C05481=1213.407,-44.587,-40.105,179.917,5.444,148.977
C05482=1213.412,-44.836,-40.092,179.914,5.443,148.977
C05483=1213.418,-45.086,-40.080,179.911,5.443,148.978
C05484=1213.422,-45.336,-40.067,179.909,5.443,148.979
C05485=1213.428,-45.586,-40.055,179.907,5.442,148.980
C05486=1213.433,-45.835,-40.043,179.904,5.442,148.980
C05487=1213.438,-46.085,-40.030,179.902,5.442,148.981
C05488=1213.443,-46.335,-40.018,179.899,5.442,148.982
C05489=1213.449,-46.584,-40.006,179.897,5.441,148.982
C05490=1213.454,-46.834,-39.994,179.894,5.442,148.983
C05491=1213.459,-47.083,-39.981,179.892,5.441,148.984
C05492=1213.464,-47.334,-39.969,179.890,5.442,148.985
C05493=1213.469,-47.583,-39.956,179.887,5.441,148.985
C05494=1213.475,-47.833,-39.944,179.885,5.440,148.986
C05495=1213.480,-48.082,-39.932,179.883,5.441,148.986
C05496=1213.485,-48.332,-39.920,179.880,5.440,148.987
C05497=1213.490,-48.602,-39.906,179.877,5.440,148.988
C05498=1213.496,-48.872,-39.894,179.874,5.440,148.989
C05499=1213.501,-49.142,-39.881,179.872,5.440,148.989
C05500=1213.507,-49.411,-39.867,179.870,5.440,148.990
C05501=1213.512,-49.662,-39.855,179.867,5.439,148.991
C05502=1213.517,-49.911,-39.843,179.865,5.439,148.992
C05503=1213.522,-50.161,-39.831,179.862,5.439,148.992
C05504=1213.527,-50.410,-39.818,179.859,5.438,148.993
C05505=1213.533,-50.660,-39.806,179.857,5.439,148.994
C05506=1213.538,-50.909,-39.794,179.855,5.438,148.994
C05507=1213.543,-51.159,-39.782,179.853,5.438,148.995
C05508=1213.548,-51.409,-39.770,179.850,5.438,148.996
C05509=1213.553,-51.658,-39.758,179.848,5.437,148.996
C05510=1213.559,-51.908,-39.746,179.846,5.438,148.997
C05511=1213.564,-52.158,-39.733,179.843,5.437,148.998
C05512=1213.568,-52.407,-39.722,179.840,5.437,148.998
C05513=1213.574,-52.657,-39.710,179.838,5.437,148.999
C05514=1213.579,-52.906,-39.698,179.836,5.437,149.000
C05515=1213.584,-53.156,-39.686,179.834,5.437,149.000
C05516=1213.590,-53.406,-39.673,179.831,5.437,149.001
C05517=1213.594,-53.655,-39.662,179.828,5.436,149.002
C05518=1213.600,-53.905,-39.650,179.827,5.436,149.002
C05519=1213.605,-54.155,-39.637,179.824,5.436,149.003
C05520=1213.610,-54.405,-39.625,179.821,5.435,149.004
C05521=1213.616,-54.654,-39.613,179.819,5.435,149.004
C05522=1213.620,-54.903,-39.601,179.817,5.435,149.005
C05523=1213.625,-55.153,-39.590,179.814,5.435,149.006
C05524=1213.631,-55.403,-39.578,179.812,5.435,149.007
C05525=1213.636,-55.653,-39.565,179.809,5.434,149.007
C05526=1213.641,-55.902,-39.554,179.807,5.435,149.008
C05527=1213.646,-56.152,-39.542,179.804,5.434,149.009
C05528=1213.651,-56.402,-39.529,179.802,5.435,149.009
C05529=1213.656,-56.651,-39.518,179.800,5.434,149.010
C05530=1213.661,-56.901,-39.506,179.797,5.433,149.011
C05531=1213.667,-57.151,-39.494,179.795,5.434,149.011
C05532=1213.672,-57.400,-39.482,179.793,5.433,149.012
C05533=1213.677,-57.650,-39.470,179.791,5.434,149.013
C05534=1213.682,-57.900,-39.459,179.788,5.433,149.013
C05535=1213.687,-58.150,-39.447,179.785,5.433,149.014
C05536=1213.692,-58.399,-39.435,179.783,5.433,149.015
C05537=1213.697,-58.649,-39.423,179.781,5.433,149.015
C05538=1213.703,-58.899,-39.411,179.778,5.433,149.016
C05539=1213.707,-59.148,-39.400,179.776,5.432,149.017
C05540=1213.713,-59.398,-39.388,179.773,5.432,149.018
C05541=1213.718,-59.648,-39.375,179.771,5.432,149.018
C05542=1213.723,-59.897,-39.364,179.769,5.432,149.019
C05543=1213.728,-60.147,-39.352,179.767,5.432,149.019
C05544=1213.734,-60.396,-39.340,179.764,5.431,149.020
C05545=1213.739,-60.646,-39.329,179.761,5.431,149.021
C05546=1213.744,-60.896,-39.317,179.759,5.431,149.022
C05547=1213.749,-61.145,-39.305,179.757,5.431,149.022
C05548=1213.754,-61.395,-39.293,179.755,5.431,149.023
C05549=1213.759,-61.645,-39.281,179.752,5.431,149.024
C05550=1213.764,-61.895,-39.270,179.749,5.430,149.024
C05551=1213.770,-62.144,-39.258,179.747,5.431,149.025
C05552=1213.775,-62.394,-39.246,179.744,5.430,149.026
C05553=1213.780,-62.644,-39.235,179.743,5.430,149.026
C05554=1213.786,-62.893,-39.224,179.740,5.430,149.027
C05555=1213.790,-63.143,-39.212,179.738,5.429,149.028
C05556=1213.796,-63.392,-39.200,179.735,5.430,149.028
C05557=1213.801,-63.642,-39.188,179.733,5.429,149.029
C05558=1213.806,-63.892,-39.176,179.731,5.429,149.030
C05559=1213.811,-64.142,-39.165,179.728,5.429,149.031
C05560=1213.816,-64.391,-39.153,179.725,5.429,149.031
C05561=1213.821,-64.641,-39.141,179.723,5.429,149.032
C05562=1213.827,-64.890,-39.131,179.721,5.428,149.033
C05563=1213.832,-65.140,-39.119,179.719,5.428,149.033
C05564=1213.837,-65.390,-39.107,179.716,5.428,149.034
C05565=1213.842,-65.640,-39.095,179.714,5.428,149.035
C05566=1213.848,-65.890,-39.084,179.712,5.428,149.035
C05567=1213.852,-66.139,-39.072,179.709,5.427,149.036
C05568=1213.858,-66.389,-39.060,179.707,5.428,149.037
C05569=1213.863,-66.638,-39.049,179.704,5.427,149.037
C05570=1213.868,-66.888,-39.038,179.702,5.428,149.038
C05571=1213.873,-67.138,-39.026,179.699,5.427,149.039
C05572=1213.878,-67.388,-39.014,179.697,5.427,149.040
C05573=1213.883,-67.637,-39.003,179.695,5.427,149.040
C05574=1213.889,-67.887,-38.991,179.692,5.426,149.041
C05575=1213.894,-68.136,-38.980,179.690,5.427,149.041
C05576=1213.899,-68.386,-38.968,179.688,5.426,149.042
C05577=1213.904,-68.636,-38.957,179.686,5.427,149.043
C05578=1213.909,-68.886,-38.945,179.683,5.426,149.044
C05579=1213.914,-69.135,-38.934,179.680,5.426,149.044
C05580=1213.920,-69.385,-38.923,179.678,5.426,149.045
C05581=1213.925,-69.635,-38.912,179.676,5.426,149.046
C05582=1213.931,-69.885,-38.900,179.673,5.426,149.046
C05583=1213.935,-70.134,-38.889,179.671,5.425,149.047
C05584=1213.941,-70.384,-38.877,179.669,5.425,149.048
C05585=1213.946,-70.633,-38.866,179.667,5.425,149.048
C05586=1213.951,-70.883,-38.855,179.664,5.425,149.049
C05587=1213.956,-71.133,-38.843,179.662,5.425,149.050
C05588=1213.961,-71.383,-38.832,179.659,5.424,149.050
C05589=1213.967,-71.632,-38.821,179.657,5.425,149.051
C05590=1213.972,-71.882,-38.809,179.654,5.424,149.052
C05591=1213.977,-72.132,-38.797,179.652,5.425,149.052
C05592=1213.982,-72.381,-38.786,179.650,5.424,149.053
C05593=1213.987,-72.630,-38.775,179.647,5.423,149.054
C05594=1213.993,-72.881,-38.764,179.645,5.424,149.054
C05595=1213.998,-73.130,-38.753,179.643,5.423,149.055
C05596=1214.003,-73.380,-38.741,179.641,5.424,149.056
C05597=1214.008,-73.629,-38.730,179.638,5.423,149.056
C05598=1214.013,-73.879,-38.719,179.636,5.424,149.057
C05599=1214.019,-74.129,-38.707,179.633,5.423,149.058
C05600=1214.024,-74.379,-38.696,179.631,5.424,149.059
C05601=1214.030,-74.649,-38.684,179.628,5.423,149.059
C05602=1214.035,-74.920,-38.671,179.626,5.423,149.060
C05603=1214.041,-75.190,-38.659,179.623,5.422,149.061
C05604=1214.046,-75.461,-38.648,179.621,5.423,149.061
C05605=1214.052,-75.711,-38.636,179.618,5.422,149.062
C05606=1214.057,-75.960,-38.626,179.616,5.422,149.063
C05607=1214.062,-76.210,-38.614,179.613,5.422,149.064
C05608=1214.067,-76.460,-38.603,179.611,5.422,149.064
C05609=1214.072,-76.709,-38.591,179.609,5.422,149.065
C05610=1214.078,-76.959,-38.581,179.607,5.421,149.065
C05611=1214.083,-77.209,-38.569,179.604,5.421,149.066
C05612=1214.088,-77.458,-38.558,179.602,5.421,149.067
C05613=1214.093,-77.708,-38.548,179.600,5.421,149.068
C05614=1214.099,-77.958,-38.536,179.597,5.421,149.068
C05615=1214.103,-78.208,-38.524,179.595,5.421,149.069
C05616=1214.109,-78.457,-38.514,179.592,5.421,149.070
C05617=1214.114,-78.707,-38.502,179.590,5.421,149.070
C05618=1214.119,-78.957,-38.491,179.588,5.420,149.071
C05619=1214.125,-79.206,-38.481,179.585,5.420,149.072
C05620=1214.129,-79.456,-38.470,179.583,5.420,149.072
C05621=1214.135,-79.706,-38.458,179.581,5.420,149.073
C05622=1214.140,-79.955,-38.447,179.579,5.420,149.074
C05623=1214.145,-80.205,-38.436,179.576,5.420,149.074
C05624=1214.150,-80.455,-38.426,179.574,5.420,149.075
C05625=1214.156,-80.704,-38.414,179.571,5.420,149.076
C05626=1214.161,-80.954,-38.403,179.569,5.420,149.076
C05627=1214.166,-81.204,-38.392,179.567,5.419,149.077
C05628=1214.171,-81.453,-38.381,179.565,5.420,149.078
C05629=1214.177,-81.704,-38.370,179.562,5.419,149.078
C05630=1214.182,-81.953,-38.359,179.559,5.419,149.079
C05631=1214.187,-82.203,-38.349,179.557,5.419,149.080
C05632=1214.192,-82.453,-38.337,179.555,5.419,149.081
C05633=1214.198,-82.702,-38.327,179.553,5.419,149.081
C05634=1214.203,-82.952,-38.315,179.550,5.418,149.082
C05635=1214.208,-83.202,-38.305,179.548,5.419,149.083
C05636=1214.213,-83.451,-38.294,179.546,5.418,149.083
C05637=1214.218,-83.701,-38.282,179.543,5.419,149.084
C05638=1214.224,-83.950,-38.272,179.541,5.418,149.085
C05639=1214.228,-84.200,-38.261,179.539,5.418,149.085
C05640=1214.234,-84.451,-38.250,179.536,5.418,149.086
C05641=1214.239,-84.699,-38.239,179.534,5.418,149.087
C05642=1214.244,-84.950,-38.228,179.532,5.418,149.087
C05643=1214.250,-85.199,-38.218,179.530,5.418,149.088
C05644=1214.255,-85.449,-38.207,179.527,5.417,149.089
C05645=1214.260,-85.699,-38.196,179.524,5.417,149.089
C05646=1214.265,-85.948,-38.185,179.522,5.417,149.090
C05647=1214.271,-86.199,-38.174,179.520,5.417,149.091
C05648=1214.276,-86.448,-38.163,179.518,5.417,149.092
C05649=1214.281,-86.698,-38.153,179.515,5.417,149.092
C05650=1214.286,-86.947,-38.142,179.513,5.417,149.093
C05651=1214.291,-87.197,-38.131,179.511,5.416,149.093
C05652=1214.296,-87.447,-38.121,179.508,5.417,149.094
C05653=1214.301,-87.696,-38.110,179.506,5.416,149.095
C05654=1214.306,-87.946,-38.099,179.504,5.417,149.096
C05655=1214.312,-88.195,-38.088,179.501,5.416,149.096
C05656=1214.317,-88.446,-38.078,179.499,5.416,149.097
C05657=1214.323,-88.695,-38.067,179.497,5.416,149.097
C05658=1214.328,-88.945,-38.055,179.495,5.416,149.098
C05659=1214.333,-89.195,-38.045,179.492,5.416,149.099
C05660=1214.338,-89.445,-38.035,179.490,5.416,149.100
C05661=1214.344,-89.694,-38.024,179.487,5.416,149.100
C05662=1214.349,-89.944,-38.013,179.485,5.416,149.101
C05663=1214.354,-90.194,-38.003,179.483,5.415,149.101
C05664=1214.359,-90.443,-37.992,179.480,5.415,149.102
C05665=1214.365,-90.693,-37.981,179.478,5.415,149.103
C05666=1214.370,-90.943,-37.971,179.476,5.415,149.104
C05667=1214.374,-91.193,-37.960,179.473,5.415,149.104
C05668=1214.380,-91.442,-37.949,179.471,5.415,149.105
C05669=1214.385,-91.692,-37.939,179.469,5.415,149.106
C05670=1214.390,-91.941,-37.928,179.466,5.414,149.106
C05671=1214.396,-92.191,-37.918,179.464,5.415,149.107
C05672=1214.401,-92.441,-37.907,179.462,5.414,149.108
C05673=1214.406,-92.691,-37.897,179.460,5.415,149.108
C05674=1214.411,-92.940,-37.886,179.457,5.414,149.109
C05675=1214.417,-93.190,-37.875,179.455,5.415,149.110
C05676=1214.422,-93.440,-37.865,179.453,5.414,149.110
C05677=1214.427,-93.690,-37.855,179.451,5.414,149.111
C05678=1214.432,-93.939,-37.843,179.448,5.414,149.112
C05679=1214.437,-94.189,-37.833,179.446,5.414,149.112
C05680=1214.442,-94.439,-37.823,179.443,5.414,149.113
C05681=1214.448,-94.689,-37.812,179.441,5.414,149.114
C05682=1214.453,-94.939,-37.802,179.439,5.413,149.114
C05683=1214.458,-95.188,-37.791,179.437,5.414,149.115
C05684=1214.463,-95.438,-37.780,179.434,5.413,149.116
C05685=1214.469,-95.687,-37.770,179.432,5.413,149.116
C05686=1214.475,-95.937,-37.760,179.429,5.413,149.117
C05687=1214.480,-96.187,-37.749,179.427,5.413,149.118
C05688=1214.485,-96.436,-37.738,179.425,5.413,149.118
C05689=1214.490,-96.686,-37.728,179.423,5.413,149.119
C05690=1214.495,-96.936,-37.718,179.420,5.413,149.120
C05691=1214.500,-97.186,-37.708,179.418,5.413,149.121
C05692=1214.505,-97.435,-37.697,179.416,5.413,149.121
C05693=1214.511,-97.685,-37.687,179.413,5.413,149.122
C05694=1214.516,-97.935,-37.677,179.411,5.412,149.122
C05695=1214.521,-98.185,-37.666,179.409,5.412,149.123
C05696=1214.526,-98.434,-37.655,179.407,5.412,149.124
C05697=1214.532,-98.684,-37.645,179.404,5.412,149.125
C05698=1214.537,-98.934,-37.635,179.402,5.412,149.125
C05699=1214.542,-99.184,-37.624,179.400,5.412,149.126
C05700=1214.547,-99.433,-37.615,179.397,5.412,149.126
C05701=1214.552,-99.683,-37.604,179.395,5.412,149.127
C05702=1214.558,-99.933,-37.594,179.393,5.411,149.128
C05703=1214.563,-100.182,-37.584,179.391,5.412,149.129
C05704=1214.568,-100.433,-37.573,179.388,5.411,149.129
C05705=1214.574,-100.704,-37.562,179.385,5.411,149.130
C05706=1214.580,-100.975,-37.551,179.383,5.411,149.131
C05707=1214.585,-101.246,-37.540,179.380,5.411,149.131
C05708=1214.591,-101.518,-37.528,179.378,5.411,149.132
C05709=1214.596,-101.767,-37.519,179.376,5.411,149.133
C05710=1214.601,-102.016,-37.508,179.374,5.411,149.134
C05711=1214.606,-102.266,-37.497,179.371,5.410,149.134
C05712=1214.612,-102.516,-37.487,179.369,5.411,149.135
C05713=1214.617,-102.766,-37.476,179.367,5.410,149.136
C05714=1214.622,-103.016,-37.468,179.365,5.411,149.136
C05715=1214.628,-103.265,-37.457,179.362,5.410,149.137
C05716=1214.633,-103.515,-37.447,179.360,5.410,149.137
C05717=1214.638,-103.765,-37.437,179.358,5.410,149.138
C05718=1214.644,-104.015,-37.426,179.356,5.410,149.139
C05719=1214.648,-104.265,-37.416,179.353,5.410,149.140
C05720=1214.654,-104.514,-37.406,179.351,5.410,149.140
C05721=1214.659,-104.764,-37.396,179.349,5.409,149.141
C05722=1214.664,-105.014,-37.385,179.347,5.410,149.141
C05723=1214.669,-105.263,-37.376,179.344,5.409,149.142
C05724=1214.675,-105.513,-37.366,179.342,5.410,149.143
C05725=1214.680,-105.763,-37.355,179.339,5.409,149.144
C05726=1214.685,-106.012,-37.345,179.337,5.409,149.144
C05727=1214.690,-106.262,-37.335,179.335,5.409,149.145
C05728=1214.696,-106.511,-37.325,179.333,5.409,149.146
C05729=1214.701,-106.762,-37.315,179.330,5.409,149.146
C05730=1214.707,-107.012,-37.305,179.328,5.409,149.147
C05731=1214.712,-107.261,-37.295,179.326,5.409,149.147
C05732=1214.717,-107.511,-37.285,179.324,5.409,149.148
C05733=1214.722,-107.761,-37.275,179.321,5.408,149.149
C05734=1214.727,-108.010,-37.265,179.319,5.409,149.150
C05735=1214.732,-108.260,-37.254,179.316,5.408,149.150
C05736=1214.738,-108.510,-37.245,179.315,5.408,149.151
C05737=1214.743,-108.759,-37.235,179.312,5.408,149.152
C05738=1214.748,-109.009,-37.225,179.310,5.408,149.152
C05739=1214.753,-109.259,-37.214,179.307,5.408,149.153
C05740=1214.759,-109.509,-37.204,179.305,5.408,149.154
C05741=1214.764,-109.758,-37.195,179.303,5.408,149.154
C05742=1214.770,-110.008,-37.185,179.301,5.408,149.155
C05743=1214.775,-110.258,-37.175,179.299,5.408,149.156
C05744=1214.780,-110.508,-37.165,179.296,5.408,149.156
C05745=1214.785,-110.757,-37.155,179.294,5.408,149.157
C05746=1214.790,-111.007,-37.146,179.292,5.407,149.157
C05747=1214.795,-111.257,-37.135,179.290,5.408,149.158
C05748=1214.801,-111.507,-37.125,179.287,5.407,149.159
C05749=1214.806,-111.756,-37.115,179.285,5.408,149.160
C05750=1214.812,-112.006,-37.106,179.283,5.407,149.160
C05751=1214.817,-112.257,-37.095,179.281,5.407,149.161
C05752=1214.822,-112.506,-37.086,179.278,5.407,149.162
C05753=1214.827,-112.755,-37.076,179.276,5.407,149.162
C05754=1214.832,-113.005,-37.067,179.273,5.407,149.163
C05755=1214.838,-113.255,-37.056,179.272,5.407,149.163
C05756=1214.843,-113.505,-37.046,179.269,5.407,149.164
C05757=1214.848,-113.755,-37.037,179.267,5.407,149.165
C05758=1214.854,-114.004,-37.027,179.264,5.407,149.166
C05759=1214.859,-114.254,-37.017,179.263,5.406,149.166
C05760=1214.864,-114.503,-37.007,179.260,5.406,149.167
C05761=1214.870,-114.754,-36.997,179.258,5.406,149.168
C05762=1214.874,-115.003,-36.987,179.255,5.406,149.168
C05763=1214.880,-115.253,-36.977,179.253,5.406,149.169
C05764=1214.885,-115.503,-36.968,179.251,5.406,149.169
C05765=1214.891,-115.752,-36.958,179.249,5.406,149.170
C05766=1214.895,-116.003,-36.949,179.247,5.406,149.171
C05767=1214.901,-116.252,-36.939,179.244,5.406,149.172
C05768=1214.907,-116.502,-36.928,179.242,5.406,149.172
C05769=1214.912,-116.752,-36.920,179.240,5.406,149.173
C05770=1214.917,-117.001,-36.909,179.238,5.406,149.173
C05771=1214.922,-117.250,-36.900,179.235,5.406,149.174
C05772=1214.927,-117.501,-36.890,179.233,5.406,149.175
C05773=1214.932,-117.750,-36.880,179.231,5.405,149.175
C05774=1214.938,-118.001,-36.871,179.229,5.406,149.176
C05775=1214.943,-118.250,-36.861,179.226,5.405,149.177
C05776=1214.949,-118.500,-36.852,179.224,5.405,149.177
C05777=1214.954,-118.749,-36.842,179.222,5.405,149.178
C05778=1214.959,-118.999,-36.832,179.219,5.405,149.179
C05779=1214.964,-119.249,-36.823,179.217,5.405,149.179
C05780=1214.970,-119.499,-36.812,179.215,5.405,149.180
C05781=1214.975,-119.749,-36.803,179.213,5.405,149.181
C05782=1214.980,-119.998,-36.793,179.210,5.405,149.181
C05783=1214.986,-120.248,-36.784,179.208,5.405,149.182
C05784=1214.990,-120.497,-36.775,179.206,5.404,149.183
C05785=1214.996,-120.748,-36.765,179.204,5.405,149.183
C05786=1215.001,-120.997,-36.755,179.201,5.404,149.184
C05787=1215.007,-121.248,-36.746,179.199,5.405,149.185
C05788=1215.011,-121.497,-36.736,179.197,5.404,149.185
C05789=1215.017,-121.747,-36.727,179.195,5.404,149.186
C05790=1215.022,-121.996,-36.717,179.192,5.404,149.187
C05791=1215.028,-122.246,-36.708,179.190,5.404,149.187
C05792=1215.033,-122.496,-36.698,179.189,5.404,149.188
C05793=1215.038,-122.746,-36.689,179.186,5.404,149.189
C05794=1215.044,-122.995,-36.679,179.184,5.404,149.189
C05795=1215.049,-123.245,-36.670,179.181,5.404,149.190
C05796=1215.054,-123.495,-36.659,179.180,5.404,149.190
C05797=1215.059,-123.745,-36.650,179.177,5.403,149.191
C05798=1215.064,-123.995,-36.642,179.175,5.404,149.192
C05799=1215.070,-124.244,-36.631,179.172,5.403,149.193
C05800=1215.075,-124.494,-36.622,179.171,5.403,149.193
C05801=1215.081,-124.744,-36.612,179.168,5.403,149.194
C05802=1215.086,-124.994,-36.603,179.166,5.403,149.195
C05803=1215.091,-125.244,-36.594,179.164,5.403,149.195
C05804=1215.096,-125.493,-36.584,179.161,5.403,149.196
C05805=1215.102,-125.743,-36.575,179.159,5.403,149.196
C05806=1215.106,-125.992,-36.566,179.157,5.403,149.197
C05807=1215.112,-126.242,-36.556,179.155,5.403,149.198
C05808=1215.118,-126.492,-36.547,179.152,5.403,149.198
C05809=1214.696,-126.503,-36.584,179.148,5.406,149.201
C05810=1214.691,-126.254,-36.593,179.151,5.406,149.200
C05811=1214.685,-126.003,-36.603,179.153,5.406,149.199
C05812=1214.680,-125.754,-36.612,179.155,5.406,149.198
C05813=1214.674,-125.504,-36.622,179.157,5.406,149.198
C05814=1214.669,-125.254,-36.631,179.160,5.407,149.197
C05815=1214.664,-125.005,-36.640,179.162,5.407,149.196
C05816=1214.658,-124.755,-36.650,179.164,5.406,149.196
C05817=1214.654,-124.504,-36.659,179.166,5.407,149.195
C05818=1214.649,-124.255,-36.669,179.168,5.407,149.195
C05819=1214.643,-124.005,-36.678,179.171,5.407,149.194
C05820=1214.638,-123.756,-36.688,179.172,5.407,149.193
C05821=1214.632,-123.506,-36.697,179.175,5.407,149.193
C05822=1214.627,-123.256,-36.706,179.177,5.407,149.192
C05823=1214.622,-123.006,-36.716,179.180,5.407,149.191
C05824=1214.616,-122.756,-36.725,179.181,5.407,149.191
C05825=1214.611,-122.507,-36.735,179.184,5.408,149.190
C05826=1214.606,-122.257,-36.745,179.186,5.407,149.189
C05827=1214.601,-122.008,-36.754,179.188,5.407,149.189
C05828=1214.596,-121.758,-36.763,179.191,5.408,149.188
C05829=1214.591,-121.508,-36.774,179.193,5.407,149.187
C05830=1214.585,-121.258,-36.783,179.195,5.408,149.187
C05831=1214.580,-121.008,-36.793,179.197,5.407,149.186
C05832=1214.575,-120.758,-36.802,179.200,5.408,149.185
C05833=1214.569,-120.509,-36.812,179.202,5.408,149.185
C05834=1214.564,-120.259,-36.821,179.204,5.408,149.184
C05835=1214.558,-120.009,-36.831,179.206,5.408,149.183
C05836=1214.553,-119.760,-36.840,179.209,5.409,149.183
C05837=1214.548,-119.509,-36.850,179.211,5.408,149.182
C05838=1214.543,-119.259,-36.859,179.213,5.409,149.181
C05839=1214.537,-119.010,-36.870,179.215,5.409,149.181
C05840=1214.532,-118.760,-36.878,179.217,5.408,149.180
C05841=1214.527,-118.511,-36.888,179.220,5.409,149.179
C05842=1214.521,-118.261,-36.898,179.222,5.408,149.179
C05843=1214.516,-118.011,-36.907,179.225,5.409,149.178
C05844=1214.511,-117.761,-36.918,179.226,5.409,149.178
C05845=1214.506,-117.511,-36.927,179.229,5.409,149.177
C05846=1214.501,-117.262,-36.937,179.231,5.409,149.176
C05847=1214.495,-117.012,-36.946,179.234,5.409,149.175
C05848=1214.490,-116.762,-36.956,179.235,5.409,149.175
C05849=1214.484,-116.513,-36.966,179.238,5.410,149.174
C05850=1214.480,-116.262,-36.975,179.240,5.409,149.173
C05851=1214.474,-116.013,-36.986,179.243,5.410,149.173
C05852=1214.469,-115.763,-36.995,179.244,5.410,149.172
C05853=1214.463,-115.513,-37.005,179.247,5.410,149.172
C05854=1214.459,-115.264,-37.014,179.249,5.410,149.171
C05855=1214.453,-115.014,-37.024,179.251,5.409,149.170
C05856=1214.448,-114.764,-37.034,179.253,5.410,149.170
C05857=1214.443,-114.514,-37.044,179.255,5.410,149.169
C05858=1214.437,-114.264,-37.053,179.258,5.410,149.168
C05859=1214.432,-114.015,-37.063,179.260,5.410,149.167
C05860=1214.426,-113.766,-37.073,179.262,5.410,149.167
C05861=1214.422,-113.515,-37.083,179.264,5.410,149.166
C05862=1214.416,-113.265,-37.093,179.267,5.410,149.166
C05863=1214.411,-113.016,-37.103,179.269,5.410,149.165
C05864=1214.406,-112.767,-37.113,179.272,5.411,149.164
C05865=1214.400,-112.516,-37.122,179.273,5.411,149.164
C05866=1214.396,-112.267,-37.132,179.276,5.411,149.163
C05867=1214.390,-112.017,-37.142,179.278,5.411,149.162
C05868=1214.384,-111.767,-37.152,179.281,5.411,149.161
C05869=1214.379,-111.518,-37.161,179.283,5.411,149.161
C05870=1214.374,-111.267,-37.172,179.285,5.411,149.160
C05871=1214.369,-111.018,-37.182,179.287,5.411,149.160
C05872=1214.364,-110.769,-37.192,179.290,5.411,149.159
C05873=1214.358,-110.518,-37.201,179.292,5.411,149.158
C05874=1214.354,-110.268,-37.211,179.294,5.412,149.158
C05875=1214.348,-110.019,-37.221,179.296,5.411,149.157
C05876=1214.342,-109.769,-37.232,179.298,5.411,149.156
C05877=1214.337,-109.520,-37.241,179.301,5.411,149.156
C05878=1214.332,-109.269,-37.251,179.303,5.412,149.155
C05879=1214.327,-109.020,-37.261,179.305,5.412,149.154
C05880=1214.322,-108.771,-37.271,179.307,5.412,149.154
C05881=1214.316,-108.521,-37.281,179.310,5.412,149.153
C05882=1214.311,-108.271,-37.292,179.312,5.412,149.152
C05883=1214.305,-108.021,-37.301,179.314,5.412,149.152
C05884=1214.301,-107.771,-37.311,179.317,5.412,149.151
C05885=1214.295,-107.522,-37.321,179.319,5.412,149.150
C05886=1214.290,-107.272,-37.332,179.321,5.412,149.150
C05887=1214.285,-107.022,-37.341,179.324,5.412,149.149
C05888=1214.279,-106.773,-37.351,179.326,5.412,149.148
C05889=1214.274,-106.523,-37.362,179.328,5.413,149.148
C05890=1214.269,-106.272,-37.372,179.330,5.413,149.147
C05891=1214.264,-106.023,-37.381,179.333,5.413,149.146
C05892=1214.259,-105.773,-37.392,179.335,5.413,149.145
C05893=1214.253,-105.523,-37.402,179.337,5.413,149.145
C05894=1214.248,-105.274,-37.412,179.339,5.413,149.144
C05895=1214.243,-105.024,-37.422,179.342,5.413,149.144
C05896=1214.238,-104.774,-37.432,179.344,5.413,149.143
C05897=1214.232,-104.525,-37.443,179.347,5.413,149.142
C05898=1214.227,-104.276,-37.452,179.348,5.413,149.142
C05899=1214.222,-104.025,-37.463,179.351,5.414,149.141
C05900=1214.217,-103.776,-37.473,179.353,5.413,149.140
C05901=1214.211,-103.526,-37.483,179.356,5.414,149.140
C05902=1214.206,-103.276,-37.494,179.358,5.414,149.139
C05903=1214.201,-103.027,-37.503,179.360,5.414,149.138
C05904=1214.196,-102.776,-37.513,179.362,5.414,149.138
C05905=1214.190,-102.526,-37.523,179.365,5.414,149.137
C05906=1214.185,-102.277,-37.534,179.367,5.414,149.136
C05907=1214.180,-102.027,-37.544,179.370,5.414,149.135
C05908=1214.175,-101.777,-37.554,179.372,5.414,149.135
C05909=1214.169,-101.528,-37.564,179.374,5.415,149.134
C05910=1214.164,-101.257,-37.576,179.376,5.414,149.134
C05911=1214.158,-100.986,-37.587,179.379,5.415,149.133
C05912=1214.152,-100.715,-37.598,179.381,5.415,149.132
C05913=1214.147,-100.443,-37.609,179.384,5.415,149.131
C05914=1214.142,-100.193,-37.620,179.386,5.415,149.131
C05915=1214.136,-99.944,-37.630,179.388,5.415,149.130
C05916=1214.130,-99.694,-37.640,179.391,5.415,149.129
C05917=1214.126,-99.444,-37.650,179.393,5.415,149.129
C05918=1214.121,-99.195,-37.660,179.396,5.415,149.128
C05919=1214.116,-98.944,-37.671,179.397,5.415,149.127
C05920=1214.110,-98.695,-37.681,179.400,5.416,149.127
C05921=1214.104,-98.445,-37.691,179.402,5.416,149.126
C05922=1214.099,-98.195,-37.702,179.405,5.416,149.125
C05923=1214.094,-97.945,-37.712,179.407,5.416,149.125
C05924=1214.089,-97.696,-37.724,179.410,5.416,149.124
C05925=1214.084,-97.447,-37.733,179.411,5.416,149.123
C05926=1214.079,-97.197,-37.743,179.414,5.416,149.123
C05927=1214.074,-96.947,-37.754,179.416,5.416,149.122
C05928=1214.068,-96.697,-37.764,179.419,5.417,149.121
C05929=1214.063,-96.447,-37.775,179.421,5.416,149.120
C05930=1214.057,-96.197,-37.785,179.423,5.417,149.120
C05931=1214.053,-95.948,-37.796,179.425,5.417,149.119
C05932=1214.047,-95.698,-37.806,179.428,5.417,149.119
C05933=1214.042,-95.449,-37.817,179.430,5.417,149.118
C05934=1214.037,-95.198,-37.827,179.432,5.417,149.117
C05935=1214.031,-94.949,-37.837,179.434,5.417,149.116
C05936=1214.026,-94.699,-37.849,179.437,5.417,149.116
C05937=1214.021,-94.450,-37.859,179.439,5.417,149.115
C05938=1214.016,-94.199,-37.870,179.441,5.418,149.115
C05939=1214.010,-93.950,-37.880,179.443,5.417,149.114
C05940=1214.005,-93.700,-37.890,179.446,5.418,149.113
C05941=1214.000,-93.451,-37.901,179.448,5.417,149.112
C05942=1213.995,-93.201,-37.912,179.451,5.418,149.112
C05943=1213.989,-92.951,-37.922,179.453,5.418,149.111
C05944=1213.984,-92.701,-37.932,179.455,5.418,149.110
C05945=1213.979,-92.452,-37.944,179.457,5.418,149.110
C05946=1213.973,-92.202,-37.954,179.460,5.418,149.109
C05947=1213.968,-91.952,-37.964,179.462,5.418,149.108
C05948=1213.963,-91.702,-37.974,179.465,5.418,149.108
C05949=1213.958,-91.453,-37.986,179.466,5.418,149.107
C05950=1213.952,-91.203,-37.996,179.469,5.419,149.106
C05951=1213.947,-90.953,-38.007,179.471,5.418,149.106
C05952=1213.942,-90.704,-38.017,179.474,5.419,149.105
C05953=1213.937,-90.454,-38.028,179.476,5.419,149.104
C05954=1213.932,-90.204,-38.038,179.479,5.419,149.104
C05955=1213.927,-89.955,-38.050,179.481,5.419,149.103
C05956=1213.921,-89.705,-38.060,179.483,5.419,149.102
C05957=1213.916,-89.455,-38.070,179.485,5.420,149.102
C05958=1213.912,-89.205,-38.082,179.488,5.419,149.101
C05959=1213.906,-88.956,-38.092,179.490,5.420,149.100
C05960=1213.901,-88.706,-38.102,179.492,5.419,149.100
C05961=1213.896,-88.457,-38.113,179.495,5.420,149.099
C05962=1213.891,-88.206,-38.124,179.497,5.420,149.098
C05963=1213.885,-87.957,-38.134,179.499,5.420,149.098
C05964=1213.880,-87.707,-38.145,179.501,5.420,149.097
C05965=1213.875,-87.458,-38.156,179.504,5.420,149.096
C05966=1213.869,-87.208,-38.168,179.506,5.420,149.096
C05967=1213.864,-86.958,-38.178,179.509,5.420,149.095
C05968=1213.859,-86.708,-38.188,179.511,5.420,149.094
C05969=1213.854,-86.458,-38.200,179.513,5.421,149.094
C05970=1213.848,-86.209,-38.210,179.515,5.420,149.093
C05971=1213.844,-85.959,-38.221,179.518,5.421,149.092
C05972=1213.838,-85.710,-38.231,179.520,5.421,149.091
C05973=1213.833,-85.460,-38.243,179.523,5.421,149.091
C05974=1213.827,-85.210,-38.253,179.525,5.421,149.090
C05975=1213.822,-84.960,-38.265,179.527,5.421,149.089
C05976=1213.817,-84.710,-38.275,179.530,5.421,149.089
C05977=1213.812,-84.461,-38.285,179.532,5.422,149.088
C05978=1213.807,-84.211,-38.297,179.534,5.422,149.087
C05979=1213.802,-83.962,-38.307,179.536,5.422,149.087
C05980=1213.797,-83.712,-38.318,179.539,5.422,149.086
C05981=1213.791,-83.461,-38.329,179.541,5.422,149.085
C05982=1213.786,-83.212,-38.340,179.544,5.422,149.085
C05983=1213.781,-82.962,-38.351,179.546,5.422,149.084
C05984=1213.776,-82.713,-38.362,179.548,5.423,149.083
C05985=1213.771,-82.464,-38.373,179.551,5.423,149.083
C05986=1213.765,-82.213,-38.384,179.553,5.423,149.082
C05987=1213.760,-81.964,-38.395,179.556,5.423,149.081
C05988=1213.755,-81.714,-38.406,179.558,5.423,149.081
C05989=1213.750,-81.464,-38.417,179.560,5.423,149.080
C05990=1213.745,-81.215,-38.427,179.562,5.423,149.079
C05991=1213.739,-80.965,-38.439,179.565,5.424,149.079
C05992=1213.734,-80.715,-38.449,179.567,5.423,149.078
C05993=1213.729,-80.466,-38.461,179.569,5.424,149.077
C05994=1213.724,-80.216,-38.472,179.571,5.423,149.077
C05995=1213.718,-79.966,-38.483,179.574,5.424,149.076
C05996=1213.713,-79.717,-38.494,179.576,5.423,149.075
C05997=1213.708,-79.466,-38.505,179.579,5.424,149.074
C05998=1213.703,-79.217,-38.516,179.581,5.424,149.074
C05999=1213.697,-78.967,-38.527,179.583,5.424,149.073
C06000=1213.692,-78.717,-38.538,179.586,5.425,149.073
C06001=1213.687,-78.468,-38.549,179.588,5.424,149.072
C06002=1213.682,-78.219,-38.560,179.591,5.425,149.071
C06003=1213.677,-77.968,-38.571,179.593,5.424,149.070
C06004=1213.671,-77.719,-38.582,179.595,5.425,149.070
C06005=1213.667,-77.470,-38.594,179.597,5.425,149.069
C06006=1213.661,-77.219,-38.605,179.600,5.425,149.068
C06007=1213.656,-76.970,-38.616,179.602,5.426,149.068
C06008=1213.651,-76.720,-38.627,179.604,5.425,149.067
C06009=1213.645,-76.470,-38.638,179.607,5.426,149.066
C06010=1213.641,-76.220,-38.649,179.609,5.426,149.066
C06011=1213.635,-75.971,-38.660,179.612,5.426,149.065
C06012=1213.630,-75.721,-38.672,179.614,5.426,149.064
C06013=1213.625,-75.471,-38.683,179.616,5.426,149.064
C06014=1213.619,-75.201,-38.695,179.619,5.426,149.063
C06015=1213.613,-74.930,-38.708,179.621,5.426,149.062
C06016=1213.608,-74.660,-38.719,179.624,5.427,149.061
C06017=1213.602,-74.390,-38.731,179.627,5.427,149.061
C06018=1213.597,-74.140,-38.743,179.629,5.427,149.060
C06019=1213.592,-73.890,-38.754,179.631,5.427,149.059
C06020=1213.586,-73.640,-38.765,179.633,5.427,149.059
C06021=1213.581,-73.391,-38.777,179.636,5.427,149.058
C06022=1213.576,-73.141,-38.788,179.638,5.427,149.057
C06023=1213.572,-72.891,-38.799,179.641,5.427,149.056
C06024=1213.566,-72.642,-38.811,179.643,5.428,149.056
C06025=1213.561,-72.392,-38.821,179.645,5.428,149.055
C06026=1213.555,-72.142,-38.833,179.648,5.428,149.055
C06027=1213.551,-71.892,-38.844,179.650,5.428,149.054
C06028=1213.545,-71.643,-38.856,179.653,5.428,149.053
C06029=1213.540,-71.393,-38.867,179.655,5.428,149.052
C06030=1213.535,-71.144,-38.878,179.657,5.428,149.052
C06031=1213.529,-70.893,-38.890,179.660,5.429,149.051
C06032=1213.524,-70.644,-38.901,179.662,5.428,149.050
C06033=1213.519,-70.394,-38.912,179.664,5.429,149.050
C06034=1213.514,-70.145,-38.924,179.666,5.429,149.049
C06035=1213.509,-69.895,-38.936,179.669,5.429,149.048
C06036=1213.503,-69.646,-38.947,179.671,5.429,149.048
C06037=1213.498,-69.396,-38.958,179.674,5.429,149.047
C06038=1213.493,-69.146,-38.970,179.676,5.430,149.046
C06039=1213.488,-68.896,-38.980,179.679,5.430,149.046
C06040=1213.483,-68.646,-38.992,179.681,5.430,149.045
C06041=1213.477,-68.397,-39.003,179.683,5.430,149.044
C06042=1213.472,-68.147,-39.015,179.686,5.430,149.043
C06043=1213.467,-67.898,-39.026,179.688,5.430,149.043
C06044=1213.462,-67.648,-39.038,179.690,5.431,149.042
C06045=1213.457,-67.398,-39.049,179.693,5.431,149.042
C06046=1213.452,-67.148,-39.061,179.695,5.431,149.041
C06047=1213.446,-66.899,-39.072,179.698,5.431,149.040
C06048=1213.441,-66.649,-39.084,179.700,5.431,149.039
C06049=1213.436,-66.400,-39.095,179.702,5.431,149.039
C06050=1213.431,-66.150,-39.107,179.705,5.432,149.038
C06051=1213.425,-65.900,-39.119,179.707,5.431,149.037
C06052=1213.421,-65.650,-39.130,179.709,5.432,149.037
C06053=1213.415,-65.401,-39.142,179.711,5.432,149.036
C06054=1213.410,-65.151,-39.153,179.714,5.432,149.035
C06055=1213.405,-64.901,-39.165,179.716,5.432,149.035
C06056=1213.400,-64.652,-39.176,179.719,5.432,149.034
C06057=1213.394,-64.402,-39.188,179.722,5.433,149.033
C06058=1213.390,-64.152,-39.200,179.724,5.432,149.033
C06059=1213.384,-63.902,-39.212,179.726,5.433,149.032
C06060=1213.378,-63.653,-39.223,179.728,5.433,149.031
C06061=1213.374,-63.403,-39.234,179.731,5.433,149.031
C06062=1213.368,-63.153,-39.246,179.733,5.434,149.030
C06063=1213.364,-62.904,-39.258,179.735,5.434,149.029
C06064=1213.358,-62.654,-39.270,179.738,5.434,149.029
C06065=1213.354,-62.405,-39.281,179.740,5.434,149.028
C06066=1213.348,-62.155,-39.293,179.743,5.434,149.027
C06067=1213.343,-61.905,-39.305,179.745,5.435,149.027
C06068=1213.338,-61.655,-39.316,179.747,5.434,149.026
C06069=1213.332,-61.406,-39.328,179.750,5.435,149.025
C06070=1213.327,-61.156,-39.340,179.752,5.434,149.024
C06071=1213.322,-60.907,-39.351,179.755,5.435,149.024
C06072=1213.317,-60.657,-39.364,179.758,5.435,149.023
C06073=1213.312,-60.408,-39.375,179.759,5.435,149.023
C06074=1213.307,-60.158,-39.387,179.762,5.436,149.022
C06075=1213.301,-59.908,-39.399,179.764,5.435,149.021
C06076=1213.297,-59.658,-39.410,179.767,5.436,149.020
C06077=1213.291,-59.408,-39.422,179.769,5.436,149.020
C06078=1213.286,-59.159,-39.435,179.771,5.436,149.019
C06079=1213.281,-58.909,-39.446,179.774,5.436,149.018
C06080=1213.276,-58.659,-39.458,179.776,5.436,149.018
C06081=1213.271,-58.409,-39.470,179.779,5.436,149.017
C06082=1213.265,-58.160,-39.481,179.781,5.437,149.016
C06083=1213.260,-57.911,-39.493,179.783,5.437,149.015
C06084=1213.255,-57.661,-39.505,179.786,5.437,149.015
C06085=1213.250,-57.412,-39.516,179.788,5.437,149.014
C06086=1213.245,-57.162,-39.528,179.790,5.438,149.014
C06087=1213.239,-56.912,-39.541,179.793,5.438,149.013
C06088=1213.234,-56.662,-39.553,179.795,5.438,149.012
C06089=1213.229,-56.413,-39.564,179.798,5.438,149.011
C06090=1213.224,-56.163,-39.577,179.800,5.438,149.011
C06091=1213.219,-55.913,-39.589,179.803,5.438,149.010
C06092=1213.213,-55.664,-39.600,179.805,5.439,149.009
C06093=1213.209,-55.414,-39.612,179.807,5.438,149.009
C06094=1213.204,-55.165,-39.624,179.810,5.439,149.008
C06095=1213.198,-54.915,-39.636,179.812,5.439,149.007
C06096=1213.193,-54.665,-39.647,179.814,5.439,149.007
C06097=1213.188,-54.416,-39.660,179.817,5.440,149.006
C06098=1213.183,-54.166,-39.672,179.819,5.439,149.005
C06099=1213.177,-53.916,-39.684,179.822,5.440,149.005
C06100=1213.172,-53.667,-39.696,179.824,5.440,149.004
C06101=1213.168,-53.417,-39.708,179.826,5.440,149.003
C06102=1213.162,-53.167,-39.720,179.829,5.440,149.003
C06103=1213.157,-52.918,-39.732,179.831,5.440,149.002
C06104=1213.152,-52.668,-39.744,179.834,5.441,149.001
C06105=1213.147,-52.419,-39.756,179.837,5.441,149.000
C06106=1213.142,-52.169,-39.768,179.839,5.441,149.000
C06107=1213.136,-51.919,-39.780,179.841,5.442,148.999
C06108=1213.131,-51.669,-39.792,179.843,5.442,148.999
C06109=1213.126,-51.420,-39.804,179.846,5.442,148.998
C06110=1213.121,-51.170,-39.817,179.848,5.442,148.997
C06111=1213.117,-50.920,-39.829,179.850,5.442,148.996
C06112=1213.111,-50.670,-39.841,179.853,5.442,148.996
C06113=1213.106,-50.421,-39.853,179.856,5.443,148.995
C06114=1213.101,-50.171,-39.865,179.858,5.442,148.994
C06115=1213.096,-49.921,-39.878,179.860,5.443,148.994
C06116=1213.090,-49.671,-39.889,179.863,5.443,148.993
C06117=1213.085,-49.422,-39.902,179.865,5.443,148.992
C06118=1213.080,-49.152,-39.915,179.868,5.443,148.992
C06119=1213.074,-48.882,-39.928,179.870,5.444,148.991
C06120=1213.069,-48.612,-39.941,179.873,5.444,148.990
C06121=1213.063,-48.343,-39.954,179.875,5.444,148.989
C06122=1213.058,-48.093,-39.967,179.878,5.444,148.989
C06123=1213.053,-47.843,-39.979,179.881,5.445,148.988
C06124=1213.048,-47.593,-39.991,179.883,5.445,148.987
C06125=1213.042,-47.344,-40.003,179.885,5.445,148.987
C06126=1213.037,-47.094,-40.016,179.887,5.445,148.986
C06127=1213.032,-46.844,-40.028,179.890,5.445,148.985
C06128=1213.027,-46.595,-40.040,179.893,5.446,148.984
C06129=1213.021,-46.345,-40.052,179.895,5.445,148.984
C06130=1213.016,-46.096,-40.065,179.897,5.446,148.983
C06131=1213.011,-45.846,-40.077,179.900,5.447,148.983
C06132=1213.006,-45.596,-40.090,179.902,5.446,148.982
C06133=1213.001,-45.346,-40.102,179.904,5.447,148.981
C06134=1212.996,-45.097,-40.114,179.907,5.447,148.981
C06135=1212.991,-44.848,-40.126,179.909,5.447,148.980
C06136=1212.986,-44.598,-40.139,179.912,5.447,148.979
C06137=1212.981,-44.348,-40.151,179.914,5.448,148.978
C06138=1212.976,-44.099,-40.163,179.917,5.447,148.978
C06139=1212.971,-43.848,-40.176,179.919,5.448,148.977
C06140=1212.966,-43.599,-40.188,179.921,5.448,148.976
C06141=1212.960,-43.350,-40.201,179.924,5.448,148.976
C06142=1212.955,-43.100,-40.213,179.927,5.449,148.975
C06143=1212.950,-42.850,-40.225,179.928,5.449,148.974
C06144=1212.945,-42.601,-40.238,179.931,5.449,148.974
C06145=1212.939,-42.351,-40.250,179.934,5.450,148.973
C06146=1212.935,-42.101,-40.263,179.936,5.449,148.972
C06147=1212.930,-41.852,-40.275,179.938,5.450,148.972
C06148=1212.924,-41.602,-40.287,179.941,5.450,148.971
C06149=1212.919,-41.353,-40.300,179.943,5.450,148.970
C06150=1212.913,-41.103,-40.313,179.946,5.450,148.970
C06151=1212.909,-40.853,-40.326,179.948,5.451,148.969
C06152=1212.903,-40.603,-40.338,179.950,5.450,148.968
C06153=1212.898,-40.354,-40.350,179.953,5.451,148.967
C06154=1212.893,-40.104,-40.363,179.956,5.451,148.967
C06155=1212.888,-39.855,-40.376,179.958,5.451,148.966
C06156=1212.883,-39.604,-40.388,179.960,5.452,148.966
C06157=1212.878,-39.355,-40.400,179.963,5.452,148.965
C06158=1212.873,-39.106,-40.413,179.965,5.452,148.964
C06159=1212.868,-38.856,-40.426,179.967,5.452,148.963
C06160=1212.862,-38.607,-40.438,179.970,5.453,148.963
C06161=1212.858,-38.356,-40.450,179.972,5.453,148.962
C06162=1212.852,-38.107,-40.464,179.975,5.453,148.961
C06163=1212.847,-37.858,-40.476,179.977,5.454,148.961
C06164=1212.842,-37.608,-40.489,179.980,5.453,148.960
C06165=1212.837,-37.359,-40.501,179.982,5.454,148.959
C06166=1212.832,-37.108,-40.514,179.985,5.454,148.959
C06167=1212.827,-36.859,-40.526,179.987,5.454,148.958
C06168=1212.821,-36.610,-40.539,179.990,5.454,148.957
C06169=1212.816,-36.360,-40.552,179.992,5.455,148.956
C06170=1212.811,-36.110,-40.565,179.994,5.455,148.956
C06171=1212.806,-35.861,-40.578,179.997,5.455,148.955
C06172=1212.801,-35.611,-40.590,179.999,5.456,148.955
C06173=1212.795,-35.361,-40.602,-179.999,5.455,148.954
C06174=1212.791,-35.111,-40.615,-179.996,5.456,148.953
C06175=1212.786,-34.862,-40.628,-179.993,5.456,148.952
C06176=1212.780,-34.612,-40.641,-179.991,5.456,148.952
C06177=1212.775,-34.362,-40.654,-179.989,5.457,148.951
C06178=1212.770,-34.113,-40.667,-179.986,5.457,148.950
C06179=1212.765,-33.864,-40.679,-179.983,5.458,148.950
C06180=1212.760,-33.614,-40.692,-179.981,5.457,148.949
C06181=1212.755,-33.364,-40.705,-179.979,5.458,148.948
C06182=1212.750,-33.115,-40.718,-179.976,5.458,148.948
C06183=1212.745,-32.866,-40.730,-179.974,5.458,148.947
C06184=1212.740,-32.615,-40.743,-179.972,5.459,148.946
C06185=1212.734,-32.366,-40.757,-179.969,5.459,148.946
C06186=1212.729,-32.117,-40.769,-179.967,5.459,148.945
C06187=1212.724,-31.867,-40.782,-179.964,5.459,148.944
C06188=1212.719,-31.617,-40.795,-179.962,5.460,148.944
C06189=1212.714,-31.368,-40.808,-179.960,5.459,148.943
C06190=1212.708,-31.118,-40.821,-179.957,5.460,148.942
C06191=1212.704,-30.868,-40.834,-179.954,5.460,148.942
C06192=1212.699,-30.619,-40.846,-179.952,5.460,148.941
C06193=1212.693,-30.369,-40.859,-179.949,5.461,148.940
C06194=1212.688,-30.119,-40.872,-179.947,5.461,148.939
C06195=1212.683,-29.870,-40.885,-179.944,5.462,148.939
C06196=1212.678,-29.621,-40.898,-179.943,5.462,148.938
C06197=1212.673,-29.370,-40.911,-179.940,5.462,148.938
C06198=1212.668,-29.121,-40.924,-179.937,5.463,148.937
C06199=1212.663,-28.871,-40.937,-179.935,5.462,148.936
C06200=1212.657,-28.621,-40.950,-179.932,5.463,148.935
C06201=1212.652,-28.372,-40.962,-179.930,5.463,148.935
C06202=1212.648,-28.122,-40.975,-179.928,5.463,148.934
C06203=1212.642,-27.873,-40.989,-179.925,5.463,148.933
C06204=1212.637,-27.624,-41.002,-179.922,5.464,148.933
C06205=1212.632,-27.374,-41.015,-179.920,5.464,148.932
C06206=1212.627,-27.124,-41.028,-179.918,5.464,148.931
C06207=1212.622,-26.874,-41.041,-179.915,5.464,148.931
C06208=1212.617,-26.625,-41.054,-179.912,5.465,148.930
C06209=1212.611,-26.375,-41.067,-179.911,5.465,148.929
C06210=1212.607,-26.126,-41.081,-179.908,5.465,148.929
C06211=1212.602,-25.876,-41.093,-179.905,5.466,148.928
C06212=1212.597,-25.626,-41.107,-179.903,5.466,148.927
C06213=1212.591,-25.377,-41.119,-179.901,5.466,148.927
C06214=1212.586,-25.127,-41.133,-179.898,5.467,148.926
C06215=1212.581,-24.877,-41.145,-179.895,5.467,148.925
C06216=1212.576,-24.628,-41.159,-179.893,5.467,148.925
C06217=1212.571,-24.378,-41.172,-179.891,5.467,148.924
C06218=1212.566,-24.129,-41.185,-179.888,5.468,148.923
C06219=1212.561,-23.879,-41.198,-179.885,5.468,148.922
C06220=1212.556,-23.630,-41.212,-179.883,5.468,148.922
C06221=1212.551,-23.380,-41.224,-179.881,5.468,148.921
C06222=1212.545,-23.110,-41.239,-179.878,5.469,148.920
C06223=1212.539,-22.841,-41.254,-179.875,5.469,148.920
C06224=1212.534,-22.572,-41.267,-179.873,5.470,148.919
C06225=1212.528,-22.302,-41.282,-179.871,5.470,148.918
C06226=1212.524,-22.052,-41.295,-179.868,5.470,148.918
C06227=1212.518,-21.803,-41.308,-179.865,5.471,148.917
C06228=1212.514,-21.553,-41.322,-179.863,5.471,148.916
C06229=1212.508,-21.304,-41.335,-179.860,5.471,148.916
C06230=1212.503,-21.054,-41.348,-179.858,5.471,148.915
C06231=1212.498,-20.804,-41.361,-179.855,5.472,148.914
C06232=1212.493,-20.555,-41.375,-179.852,5.472,148.913
C06233=1212.487,-20.305,-41.388,-179.850,5.472,148.913
C06234=1212.483,-20.056,-41.401,-179.848,5.473,148.912
C06235=1212.477,-19.806,-41.415,-179.846,5.473,148.912
C06236=1212.472,-19.557,-41.428,-179.843,5.474,148.911
C06237=1212.467,-19.307,-41.442,-179.841,5.473,148.910
C06238=1212.462,-19.058,-41.454,-179.838,5.474,148.909
C06239=1212.457,-18.807,-41.468,-179.836,5.474,148.909
C06240=1212.452,-18.559,-41.481,-179.833,5.474,148.908
C06241=1212.447,-18.308,-41.495,-179.831,5.474,148.907
C06242=1212.442,-18.060,-41.508,-179.828,5.475,148.907
C06243=1212.437,-17.809,-41.522,-179.825,5.475,148.906
C06244=1212.432,-17.560,-41.534,-179.823,5.475,148.905
C06245=1212.427,-17.310,-41.549,-179.821,5.476,148.905
C06246=1212.421,-17.061,-41.562,-179.818,5.476,148.904
C06247=1212.417,-16.811,-41.576,-179.816,5.477,148.903
C06248=1212.411,-16.562,-41.589,-179.814,5.477,148.903
C06249=1212.407,-16.312,-41.602,-179.811,5.477,148.902
C06250=1212.401,-16.062,-41.616,-179.809,5.478,148.901
C06251=1212.396,-15.813,-41.629,-179.806,5.478,148.901
C06252=1212.391,-15.563,-41.643,-179.804,5.478,148.900
C06253=1212.386,-15.314,-41.657,-179.801,5.478,148.899
C06254=1212.381,-15.064,-41.670,-179.798,5.479,148.899
C06255=1212.376,-14.815,-41.684,-179.796,5.479,148.898
C06256=1212.371,-14.565,-41.697,-179.794,5.479,148.897
C06257=1212.365,-14.316,-41.711,-179.791,5.480,148.897
C06258=1212.360,-14.066,-41.724,-179.788,5.480,148.896
C06259=1212.356,-13.816,-41.738,-179.786,5.481,148.895
C06260=1212.350,-13.567,-41.751,-179.784,5.481,148.895
C06261=1212.345,-13.317,-41.765,-179.782,5.481,148.894
C06262=1212.340,-13.067,-41.778,-179.779,5.482,148.893
C06263=1212.335,-12.818,-41.792,-179.776,5.482,148.893
C06264=1212.330,-12.569,-41.806,-179.774,5.482,148.892
C06265=1212.325,-12.319,-41.819,-179.771,5.482,148.891
C06266=1212.320,-12.069,-41.833,-179.769,5.483,148.891
C06267=1212.314,-11.819,-41.846,-179.766,5.483,148.890
C06268=1212.310,-11.570,-41.860,-179.764,5.484,148.889
C06269=1212.304,-11.321,-41.874,-179.761,5.483,148.888
C06270=1212.299,-11.071,-41.888,-179.759,5.484,148.888
C06271=1212.295,-10.821,-41.901,-179.757,5.485,148.887
C06272=1212.289,-10.572,-41.915,-179.754,5.485,148.887
C06273=1212.284,-10.322,-41.929,-179.752,5.485,148.886
C06274=1212.280,-10.073,-41.942,-179.749,5.485,148.885
C06275=1212.274,-9.823,-41.956,-179.747,5.486,148.885
C06276=1212.269,-9.573,-41.970,-179.744,5.486,148.884
C06277=1212.264,-9.324,-41.984,-179.742,5.486,148.883
C06278=1212.259,-9.075,-41.998,-179.739,5.487,148.882
C06279=1212.254,-8.824,-42.011,-179.737,5.487,148.882
C06280=1212.249,-8.575,-42.025,-179.734,5.488,148.881
C06281=1212.244,-8.326,-42.039,-179.731,5.488,148.880
C06282=1212.239,-8.076,-42.052,-179.729,5.488,148.880
C06283=1212.233,-7.827,-42.066,-179.727,5.489,148.879
C06284=1212.229,-7.577,-42.080,-179.724,5.489,148.879
C06285=1212.224,-7.327,-42.095,-179.722,5.490,148.878
C06286=1212.218,-7.078,-42.107,-179.720,5.489,148.877
C06287=1212.214,-6.828,-42.122,-179.717,5.490,148.876
C06288=1212.209,-6.579,-42.136,-179.714,5.490,148.876
C06289=1212.203,-6.330,-42.150,-179.712,5.491,148.875
C06290=1212.198,-6.079,-42.163,-179.709,5.491,148.874
C06291=1212.194,-5.830,-42.177,-179.707,5.491,148.874
C06292=1212.188,-5.581,-42.191,-179.704,5.492,148.873
C06293=1212.183,-5.331,-42.205,-179.702,5.492,148.872
C06294=1212.178,-5.081,-42.219,-179.699,5.493,148.872
C06295=1212.173,-4.831,-42.233,-179.697,5.493,148.871
C06296=1212.167,-4.582,-42.247,-179.695,5.493,148.870
C06297=1212.163,-4.333,-42.261,-179.692,5.494,148.870
C06298=1212.158,-4.083,-42.275,-179.689,5.494,148.869
C06299=1212.153,-3.834,-42.289,-179.687,5.495,148.868
C06300=1212.148,-3.584,-42.303,-179.684,5.495,148.868
C06301=1212.143,-3.334,-42.317,-179.682,5.495,148.867
C06302=1212.137,-3.084,-42.331,-179.679,5.495,148.866
C06303=1212.132,-2.835,-42.345,-179.677,5.496,148.866
C06304=1212.128,-2.586,-42.359,-179.674,5.496,148.865
C06305=1212.123,-2.336,-42.373,-179.672,5.497,148.865
C06306=1212.118,-2.086,-42.387,-179.670,5.497,148.864
C06307=1212.112,-1.837,-42.401,-179.667,5.497,148.863
C06308=1212.107,-1.588,-42.415,-179.664,5.498,148.862
C06309=1212.102,-1.338,-42.430,-179.662,5.498,148.862
C06310=1212.097,-1.088,-42.444,-179.659,5.499,148.861
C06311=1212.092,-0.839,-42.458,-179.657,5.499,148.860
C06312=1212.087,-0.589,-42.472,-179.654,5.499,148.860
C06313=1212.082,-0.340,-42.486,-179.652,5.500,148.859
C06314=1212.077,-0.090,-42.501,-179.649,5.500,148.858
C06315=1212.072,0.159,-42.514,-179.647,5.501,148.858
C06316=1212.067,0.408,-42.528,-179.645,5.501,148.857
C06317=1212.062,0.658,-42.542,-179.642,5.501,148.856
C06318=1212.057,0.908,-42.557,-179.640,5.502,148.856
C06319=1212.052,1.157,-42.571,-179.637,5.502,148.855
C06320=1212.047,1.406,-42.585,-179.634,5.503,148.854
C06321=1212.042,1.656,-42.599,-179.632,5.503,148.854
C06322=1212.037,1.906,-42.613,-179.630,5.503,148.853
C06323=1212.032,2.156,-42.628,-179.627,5.503,148.852
C06324=1212.027,2.405,-42.642,-179.624,5.504,148.852
C06325=1212.021,2.654,-42.656,-179.622,5.505,148.851
C06326=1212.016,2.924,-42.671,-179.619,5.505,148.850
C06327=1212.011,3.193,-42.687,-179.616,5.505,148.850
C06328=1212.005,3.462,-42.702,-179.614,5.506,148.849
C06329=1211.999,3.731,-42.718,-179.611,5.506,148.848
C06330=1211.994,3.981,-42.732,-179.609,5.506,148.848
C06331=1211.989,4.230,-42.746,-179.606,5.507,148.847
C06332=1211.984,4.480,-42.760,-179.604,5.507,148.846
C06333=1211.979,4.729,-42.775,-179.601,5.508,148.845
C06334=1211.974,4.979,-42.789,-179.599,5.509,148.845
C06335=1211.969,5.228,-42.804,-179.596,5.509,148.844
C06336=1211.964,5.478,-42.818,-179.594,5.509,148.844
C06337=1211.959,5.727,-42.832,-179.591,5.509,148.843
C06338=1211.954,5.976,-42.846,-179.589,5.510,148.842
C06339=1211.949,6.226,-42.861,-179.586,5.510,148.842
C06340=1211.944,6.476,-42.875,-179.583,5.511,148.841
C06341=1211.939,6.725,-42.890,-179.581,5.511,148.840
C06342=1211.934,6.975,-42.904,-179.578,5.512,148.840
C06343=1211.929,7.225,-42.919,-179.577,5.512,148.839
C06344=1211.924,7.474,-42.933,-179.574,5.512,148.838
C06345=1211.919,7.724,-42.948,-179.571,5.513,148.838
C06346=1211.914,7.973,-42.962,-179.569,5.513,148.837
C06347=1211.909,8.222,-42.977,-179.566,5.514,148.836
C06348=1211.904,8.472,-42.991,-179.563,5.515,148.836
C06349=1211.899,8.722,-43.005,-179.561,5.514,148.835
C06350=1211.894,8.971,-43.020,-179.559,5.515,148.834
C06351=1211.888,9.221,-43.035,-179.556,5.515,148.834
C06352=1211.883,9.470,-43.049,-179.554,5.516,148.833
C06353=1211.878,9.720,-43.064,-179.551,5.517,148.832
C06354=1211.874,9.969,-43.079,-179.548,5.517,148.832
C06355=1211.869,10.219,-43.093,-179.546,5.518,148.831
C06356=1211.864,10.469,-43.107,-179.544,5.517,148.830
C06357=1211.858,10.717,-43.122,-179.541,5.518,148.830
C06358=1211.853,10.967,-43.137,-179.538,5.518,148.829
C06359=1211.848,11.217,-43.151,-179.536,5.519,148.828
C06360=1211.843,11.466,-43.166,-179.533,5.519,148.828
C06361=1211.838,11.716,-43.180,-179.531,5.520,148.827
C06362=1211.833,11.966,-43.195,-179.528,5.521,148.826
C06363=1211.828,12.215,-43.210,-179.526,5.521,148.826
C06364=1211.823,12.464,-43.224,-179.524,5.521,148.825
C06365=1211.818,12.714,-43.239,-179.521,5.522,148.824
C06366=1211.813,12.963,-43.254,-179.518,5.522,148.824
C06367=1211.808,13.213,-43.268,-179.516,5.523,148.823
C06368=1211.803,13.462,-43.283,-179.513,5.523,148.822
C06369=1211.798,13.712,-43.298,-179.510,5.524,148.822
C06370=1211.794,13.961,-43.313,-179.508,5.525,148.821
C06371=1211.788,14.211,-43.328,-179.506,5.524,148.821
C06372=1211.783,14.461,-43.342,-179.504,5.525,148.820
C06373=1211.778,14.710,-43.357,-179.501,5.525,148.819
C06374=1211.773,14.960,-43.371,-179.498,5.526,148.818
C06375=1211.768,15.209,-43.387,-179.496,5.526,148.818
C06376=1211.763,15.459,-43.401,-179.493,5.527,148.817
C06377=1211.758,15.708,-43.416,-179.490,5.527,148.816
C06378=1211.753,15.958,-43.431,-179.488,5.528,148.816
C06379=1211.748,16.207,-43.446,-179.486,5.528,148.815
C06380=1211.743,16.457,-43.460,-179.483,5.528,148.815
C06381=1211.738,16.706,-43.476,-179.481,5.529,148.814
C06382=1211.733,16.956,-43.490,-179.478,5.529,148.813
C06383=1211.728,17.205,-43.505,-179.475,5.530,148.813
C06384=1211.722,17.455,-43.520,-179.473,5.531,148.812
C06385=1211.718,17.704,-43.535,-179.470,5.531,148.811
C06386=1211.713,17.954,-43.549,-179.468,5.532,148.811
C06387=1211.707,18.203,-43.565,-179.466,5.532,148.810
C06388=1211.702,18.453,-43.579,-179.463,5.532,148.809
C06389=1211.698,18.702,-43.594,-179.461,5.533,148.809
C06390=1211.692,18.951,-43.610,-179.458,5.533,148.808
C06391=1211.687,19.201,-43.624,-179.455,5.534,148.807
C06392=1211.683,19.450,-43.639,-179.453,5.534,148.807
C06393=1211.678,19.701,-43.654,-179.451,5.535,148.806
C06394=1211.673,19.950,-43.669,-179.448,5.536,148.806
C06395=1211.668,20.199,-43.685,-179.445,5.536,148.805
C06396=1211.663,20.449,-43.699,-179.443,5.537,148.804
C06397=1211.658,20.698,-43.714,-179.441,5.536,148.803
C06398=1211.653,20.948,-43.729,-179.438,5.537,148.803
C06399=1211.648,21.197,-43.744,-179.435,5.537,148.802
C06400=1211.642,21.447,-43.759,-179.433,5.538,148.801
C06401=1211.638,21.696,-43.774,-179.430,5.539,148.801
C06402=1211.633,21.945,-43.789,-179.428,5.539,148.800
C06403=1211.627,22.195,-43.804,-179.425,5.540,148.800
C06404=1211.623,22.445,-43.820,-179.422,5.540,148.799
C06405=1211.618,22.695,-43.834,-179.420,5.541,148.798
C06406=1211.613,22.944,-43.849,-179.417,5.541,148.798
C06407=1211.607,23.193,-43.865,-179.415,5.542,148.797
C06408=1211.603,23.442,-43.880,-179.413,5.542,148.796
C06409=1211.597,23.692,-43.895,-179.410,5.543,148.796
C06410=1211.592,23.941,-43.910,-179.408,5.543,148.795
C06411=1211.587,24.191,-43.925,-179.405,5.544,148.794
C06412=1211.583,24.441,-43.941,-179.402,5.544,148.794
C06413=1211.577,24.691,-43.956,-179.400,5.545,148.793
C06414=1211.573,24.940,-43.971,-179.397,5.545,148.792
C06415=1211.567,25.189,-43.986,-179.395,5.546,148.792
C06416=1211.563,25.438,-44.001,-179.392,5.547,148.791
C06417=1211.557,25.688,-44.016,-179.390,5.547,148.791
C06418=1211.552,25.937,-44.031,-179.387,5.548,148.790
C06419=1211.548,26.187,-44.047,-179.384,5.548,148.789
C06420=1211.543,26.437,-44.062,-179.382,5.548,148.789
C06421=1211.538,26.686,-44.078,-179.380,5.548,148.788
C06422=1211.533,26.935,-44.093,-179.377,5.549,148.787
C06423=1211.527,27.185,-44.108,-179.375,5.550,148.787
C06424=1211.522,27.434,-44.123,-179.372,5.550,148.786
C06425=1211.518,27.684,-44.138,-179.370,5.551,148.785
C06426=1211.512,27.934,-44.154,-179.367,5.552,148.785
C06427=1211.508,28.183,-44.169,-179.364,5.552,148.784
C06428=1211.502,28.432,-44.185,-179.362,5.553,148.784
C06429=1211.498,28.681,-44.200,-179.359,5.553,148.783
C06430=1211.492,28.951,-44.216,-179.357,5.554,148.782
C06431=1211.487,29.219,-44.233,-179.354,5.555,148.782
C06432=1211.482,29.488,-44.250,-179.352,5.555,148.781
C06433=1211.476,29.757,-44.266,-179.348,5.555,148.780
C06434=1211.471,30.006,-44.282,-179.346,5.556,148.779
C06435=1211.466,30.255,-44.297,-179.344,5.557,148.779
C06436=1211.461,30.505,-44.312,-179.341,5.557,148.778
C06437=1211.456,30.755,-44.328,-179.338,5.558,148.777
C06438=1211.451,31.004,-44.343,-179.336,5.558,148.777
C06439=1211.446,31.253,-44.359,-179.333,5.559,148.776
C06440=1211.441,31.503,-44.374,-179.331,5.560,148.776
C06441=1211.436,31.752,-44.390,-179.328,5.560,148.775
C06442=1211.431,32.002,-44.405,-179.326,5.561,148.774
C06443=1211.426,32.251,-44.421,-179.323,5.561,148.774
C06444=1211.421,32.500,-44.436,-179.320,5.562,148.773
C06445=1211.416,32.750,-44.452,-179.318,5.562,148.772
C06446=1211.411,33.000,-44.467,-179.315,5.563,148.772
C06447=1211.406,33.249,-44.482,-179.313,5.564,148.771
C06448=1211.401,33.499,-44.498,-179.310,5.564,148.770
C06449=1211.396,33.748,-44.514,-179.308,5.564,148.770
C06450=1211.391,33.998,-44.529,-179.306,5.565,148.769
C06451=1211.386,34.247,-44.545,-179.303,5.565,148.768
C06452=1211.382,34.496,-44.561,-179.301,5.566,148.768
C06453=1211.376,34.746,-44.577,-179.298,5.567,148.767
C06454=1211.372,34.995,-44.592,-179.295,5.567,148.767
C06455=1211.367,35.245,-44.608,-179.293,5.568,148.766
C06456=1211.361,35.494,-44.623,-179.290,5.568,148.765
C06457=1211.356,35.744,-44.639,-179.287,5.569,148.765
C06458=1211.352,35.994,-44.654,-179.285,5.570,148.764
C06459=1211.347,36.243,-44.670,-179.283,5.570,148.763
C06460=1211.341,36.492,-44.686,-179.280,5.571,148.763
C06461=1211.336,36.741,-44.702,-179.277,5.571,148.762
C06462=1211.331,36.991,-44.718,-179.275,5.572,148.761
C06463=1211.327,37.240,-44.733,-179.272,5.572,148.761
C06464=1211.321,37.490,-44.748,-179.270,5.573,148.760
C06465=1211.317,37.739,-44.765,-179.267,5.574,148.760
C06466=1211.311,37.989,-44.781,-179.265,5.574,148.759
C06467=1211.306,38.238,-44.796,-179.262,5.575,148.758
C06468=1211.302,38.488,-44.811,-179.259,5.575,148.758
C06469=1211.297,38.737,-44.827,-179.257,5.576,148.757
C06470=1211.292,38.987,-44.844,-179.255,5.577,148.757
C06471=1211.287,39.236,-44.859,-179.252,5.577,148.756
C06472=1211.281,39.486,-44.875,-179.249,5.578,148.755
C06473=1211.276,39.736,-44.891,-179.247,5.578,148.755
C06474=1211.272,39.984,-44.907,-179.244,5.579,148.754
C06475=1211.267,40.234,-44.922,-179.242,5.580,148.753
C06476=1211.262,40.484,-44.938,-179.239,5.580,148.753
C06477=1211.257,40.732,-44.954,-179.237,5.581,148.752
C06478=1211.252,40.983,-44.970,-179.234,5.581,148.751
C06479=1211.247,41.232,-44.986,-179.231,5.582,148.751
C06480=1211.242,41.481,-45.002,-179.229,5.583,148.750
C06481=1211.237,41.731,-45.018,-179.227,5.583,148.750
C06482=1211.231,41.980,-45.034,-179.224,5.584,148.749
C06483=1211.227,42.230,-45.050,-179.221,5.584,148.748
C06484=1211.222,42.479,-45.065,-179.219,5.585,148.748
C06485=1211.217,42.728,-45.081,-179.216,5.586,148.747
C06486=1211.212,42.978,-45.098,-179.214,5.586,148.746
C06487=1211.207,43.227,-45.113,-179.211,5.587,148.746
C06488=1211.203,43.477,-45.130,-179.209,5.588,148.745
C06489=1211.197,43.726,-45.146,-179.206,5.588,148.744
C06490=1211.192,43.976,-45.162,-179.204,5.589,148.744
C06491=1211.187,44.225,-45.178,-179.201,5.590,148.743
C06492=1211.182,44.474,-45.193,-179.199,5.590,148.743
C06493=1211.177,44.724,-45.210,-179.196,5.591,148.742
C06494=1211.172,44.973,-45.226,-179.193,5.591,148.741
C06495=1211.168,45.223,-45.242,-179.191,5.592,148.741
C06496=1211.162,45.472,-45.258,-179.188,5.593,148.740
C06497=1211.157,45.722,-45.274,-179.186,5.593,148.740
C06498=1211.152,45.971,-45.290,-179.183,5.594,148.739
C06499=1211.148,46.221,-45.306,-179.181,5.594,148.738
C06500=1211.143,46.470,-45.322,-179.178,5.595,148.738
C06501=1211.138,46.720,-45.338,-179.176,5.596,148.737
C06502=1211.133,46.969,-45.355,-179.173,5.596,148.736
C06503=1211.128,47.219,-45.371,-179.170,5.597,148.736
C06504=1211.123,47.468,-45.387,-179.168,5.597,148.735
C06505=1211.118,47.717,-45.404,-179.166,5.598,148.735
C06506=1211.113,47.966,-45.419,-179.163,5.599,148.734
C06507=1211.108,48.216,-45.436,-179.160,5.599,148.733
C06508=1211.103,48.465,-45.451,-179.158,5.600,148.733
C06509=1211.099,48.715,-45.468,-179.155,5.600,148.732
C06510=1211.093,48.964,-45.484,-179.153,5.601,148.731
C06511=1211.089,49.214,-45.500,-179.150,5.602,148.731
C06512=1211.084,49.463,-45.517,-179.148,5.602,148.730
C06513=1211.078,49.713,-45.533,-179.144,5.604,148.729
C06514=1211.073,49.962,-45.550,-179.142,5.605,148.729
C06515=1211.068,50.212,-45.565,-179.140,5.605,148.728
C06516=1211.063,50.461,-45.582,-179.137,5.606,148.728
C06517=1211.059,50.710,-45.598,-179.134,5.606,148.727
C06518=1211.053,50.959,-45.614,-179.132,5.607,148.726
C06519=1211.049,51.209,-45.631,-179.130,5.608,148.726
C06520=1211.044,51.458,-45.647,-179.127,5.608,148.725
C06521=1211.039,51.708,-45.663,-179.124,5.609,148.725
C06522=1211.034,51.958,-45.680,-179.122,5.609,148.724
C06523=1211.029,52.206,-45.697,-179.120,5.610,148.723
C06524=1211.024,52.456,-45.713,-179.117,5.611,148.723
C06525=1211.019,52.705,-45.729,-179.114,5.611,148.722
C06526=1211.014,52.955,-45.745,-179.112,5.612,148.721
C06527=1211.010,53.204,-45.762,-179.109,5.613,148.721
C06528=1211.004,53.454,-45.778,-179.107,5.613,148.720
C06529=1210.999,53.703,-45.795,-179.104,5.614,148.720
C06530=1210.994,53.952,-45.811,-179.102,5.615,148.719
C06531=1210.990,54.202,-45.828,-179.099,5.615,148.718
C06532=1210.984,54.451,-45.844,-179.096,5.617,148.718
C06533=1210.979,54.701,-45.861,-179.094,5.617,148.717
C06534=1210.974,54.969,-45.879,-179.091,5.618,148.717
C06535=1210.969,55.238,-45.896,-179.088,5.619,148.716
C06536=1210.964,55.506,-45.914,-179.086,5.619,148.715
C06537=1210.958,55.775,-45.932,-179.083,5.620,148.715
C06538=1210.953,56.024,-45.949,-179.080,5.621,148.714
C06539=1210.948,56.274,-45.965,-179.077,5.622,148.713
C06540=1210.944,56.523,-45.981,-179.075,5.622,148.713
C06541=1210.938,56.772,-45.998,-179.072,5.623,148.712
C06542=1210.934,57.022,-46.015,-179.070,5.624,148.711
C06543=1210.929,57.271,-46.032,-179.067,5.624,148.711
C06544=1210.923,57.520,-46.048,-179.065,5.625,148.710
C06545=1210.919,57.770,-46.065,-179.062,5.626,148.710
C06546=1210.914,58.019,-46.081,-179.060,5.626,148.709
C06547=1210.909,58.269,-46.097,-179.057,5.627,148.708
C06548=1210.904,58.518,-46.115,-179.055,5.628,148.708
C06549=1210.899,58.767,-46.131,-179.052,5.628,148.707
C06550=1210.894,59.017,-46.148,-179.049,5.630,148.707
C06551=1210.889,59.266,-46.165,-179.047,5.630,148.706
C06552=1210.884,59.515,-46.181,-179.044,5.631,148.706
C06553=1210.879,59.765,-46.198,-179.042,5.632,148.705
C06554=1210.874,60.015,-46.215,-179.039,5.632,148.704
C06555=1210.870,60.264,-46.232,-179.036,5.633,148.704
C06556=1210.865,60.513,-46.248,-179.034,5.634,148.703
C06557=1210.859,60.763,-46.265,-179.032,5.634,148.702
C06558=1210.855,61.012,-46.282,-179.029,5.635,148.702
C06559=1210.850,61.261,-46.298,-179.026,5.635,148.701
C06560=1210.845,61.511,-46.316,-179.024,5.636,148.701
C06561=1210.840,61.760,-46.332,-179.021,5.638,148.700
C06562=1210.835,62.010,-46.349,-179.018,5.638,148.699
C06563=1210.830,62.259,-46.366,-179.016,5.639,148.699
C06564=1210.825,62.508,-46.382,-179.014,5.640,148.698
C06565=1210.820,62.758,-46.400,-179.011,5.640,148.698
C06566=1210.815,63.007,-46.416,-179.008,5.641,148.697
C06567=1210.810,63.257,-46.433,-179.006,5.641,148.696
C06568=1210.805,63.506,-46.450,-179.004,5.642,148.696
C06569=1210.801,63.755,-46.467,-179.001,5.643,148.695
C06570=1210.795,64.004,-46.484,-178.998,5.644,148.695
C06571=1210.791,64.254,-46.501,-178.996,5.645,148.694
C06572=1210.786,64.503,-46.518,-178.993,5.646,148.693
C06573=1210.781,64.753,-46.535,-178.990,5.646,148.693
C06574=1210.775,65.002,-46.552,-178.988,5.647,148.692
C06575=1210.771,65.251,-46.568,-178.986,5.648,148.692
C06576=1210.766,65.501,-46.586,-178.983,5.648,148.691
C06577=1210.761,65.750,-46.603,-178.980,5.649,148.690
C06578=1210.756,66.000,-46.620,-178.978,5.649,148.690
C06579=1210.751,66.249,-46.637,-178.975,5.651,148.689
C06580=1210.746,66.498,-46.654,-178.972,5.652,148.689
C06581=1210.741,66.748,-46.671,-178.970,5.652,148.688
C06582=1210.737,66.997,-46.689,-178.968,5.653,148.687
C06583=1210.732,67.247,-46.705,-178.965,5.654,148.687
C06584=1210.726,67.496,-46.722,-178.962,5.654,148.686
C06585=1210.722,67.745,-46.739,-178.960,5.655,148.685
C06586=1210.717,67.994,-46.757,-178.958,5.656,148.685
C06587=1210.712,68.244,-46.773,-178.954,5.657,148.684
C06588=1210.707,68.494,-46.791,-178.952,5.658,148.684
C06589=1210.702,68.742,-46.807,-178.950,5.659,148.683
C06590=1210.697,68.992,-46.825,-178.947,5.659,148.683
C06591=1210.693,69.241,-46.842,-178.944,5.660,148.682
C06592=1210.687,69.491,-46.859,-178.942,5.660,148.681
C06593=1210.683,69.740,-46.876,-178.940,5.661,148.681
C06594=1210.678,69.989,-46.894,-178.936,5.663,148.680
C06595=1210.673,70.239,-46.911,-178.934,5.663,148.680
C06596=1210.668,70.487,-46.928,-178.932,5.664,148.679
C06597=1210.663,70.737,-46.945,-178.929,5.665,148.678
C06598=1210.658,70.987,-46.962,-178.926,5.665,148.678
C06599=1210.653,71.236,-46.980,-178.924,5.666,148.677
C06600=1210.648,71.486,-46.997,-178.921,5.667,148.677
C06601=1210.644,71.735,-47.014,-178.918,5.668,148.676
C06602=1210.639,71.984,-47.032,-178.916,5.669,148.675
C06603=1210.634,72.234,-47.049,-178.914,5.670,148.675
C06604=1210.629,72.482,-47.066,-178.911,5.670,148.674
C06605=1210.624,72.732,-47.083,-178.908,5.671,148.674
C06606=1210.618,72.982,-47.100,-178.906,5.672,148.673
C06607=1210.614,73.231,-47.118,-178.903,5.673,148.673
C06608=1210.609,73.481,-47.135,-178.900,5.674,148.672
C06609=1210.604,73.730,-47.153,-178.898,5.674,148.671
C06610=1210.600,73.979,-47.170,-178.896,5.675,148.671
C06611=1210.595,74.228,-47.188,-178.893,5.676,148.670
C06612=1210.590,74.478,-47.205,-178.890,5.676,148.670
C06613=1210.585,74.727,-47.222,-178.888,5.678,148.669
C06614=1210.580,74.976,-47.239,-178.885,5.678,148.668
C06615=1210.575,75.225,-47.257,-178.882,5.679,148.668
C06616=1210.570,75.475,-47.274,-178.880,5.680,148.667
C06617=1210.565,75.724,-47.292,-178.878,5.681,148.667
C06618=1210.560,75.974,-47.309,-178.875,5.681,148.666
C06619=1210.555,76.223,-47.327,-178.872,5.683,148.666
C06620=1210.551,76.472,-47.344,-178.870,5.683,148.665
C06621=1210.546,76.722,-47.362,-178.867,5.684,148.664
C06622=1210.540,76.971,-47.379,-178.865,5.685,148.664
C06623=1210.536,77.221,-47.397,-178.862,5.685,148.663
C06624=1210.531,77.469,-47.414,-178.859,5.687,148.663
C06625=1210.526,77.719,-47.432,-178.857,5.688,148.662
C06626=1210.521,77.968,-47.450,-178.854,5.688,148.661
C06627=1210.516,78.218,-47.467,-178.852,5.689,148.661
C06628=1210.512,78.467,-47.484,-178.850,5.690,148.660
C06629=1210.507,78.716,-47.502,-178.846,5.691,148.660
C06630=1210.502,78.966,-47.520,-178.844,5.692,148.659
C06631=1210.497,79.215,-47.538,-178.842,5.693,148.659
C06632=1210.492,79.464,-47.556,-178.839,5.693,148.658
C06633=1210.487,79.714,-47.573,-178.836,5.694,148.657
C06634=1210.483,79.963,-47.590,-178.834,5.695,148.657
C06635=1210.478,80.212,-47.608,-178.831,5.696,148.656
C06636=1210.472,80.462,-47.625,-178.828,5.697,148.656
C06637=1210.467,80.711,-47.643,-178.826,5.698,148.655
C06638=1210.462,80.979,-47.663,-178.824,5.698,148.655
C06639=1210.457,81.248,-47.682,-178.820,5.700,148.654
C06640=1210.451,81.516,-47.701,-178.818,5.700,148.653
C06641=1210.446,81.784,-47.720,-178.815,5.702,148.653
C06642=1210.441,82.034,-47.737,-178.812,5.702,148.652
C06643=1210.436,82.283,-47.755,-178.810,5.703,148.651
C06644=1210.432,82.532,-47.773,-178.807,5.704,148.651
C06645=1210.428,82.782,-47.791,-178.805,5.704,148.650
C06646=1210.422,83.032,-47.808,-178.802,5.706,148.650
C06647=1210.417,83.281,-47.826,-178.799,5.707,148.649
C06648=1210.413,83.530,-47.844,-178.797,5.708,148.649
C06649=1210.408,83.779,-47.862,-178.795,5.708,148.648
C06650=1210.403,84.028,-47.880,-178.791,5.710,148.647
C06651=1210.398,84.278,-47.897,-178.789,5.710,148.647
C06652=1210.393,84.527,-47.915,-178.787,5.711,148.646
C06653=1210.388,84.776,-47.933,-178.784,5.712,148.646
C06654=1210.383,85.026,-47.951,-178.782,5.713,148.645
C06655=1210.378,85.275,-47.969,-178.779,5.714,148.645
C06656=1210.373,85.524,-47.987,-178.776,5.715,148.644
C06657=1210.368,85.773,-48.005,-178.774,5.715,148.644
C06658=1210.363,86.024,-48.023,-178.771,5.716,148.643
C06659=1210.359,86.273,-48.041,-178.768,5.717,148.642
C06660=1210.354,86.522,-48.059,-178.766,5.718,148.642
C06661=1210.349,86.771,-48.077,-178.763,5.719,148.641
C06662=1210.344,87.020,-48.095,-178.761,5.720,148.641
C06663=1210.339,87.270,-48.113,-178.758,5.721,148.640
C06664=1210.334,87.519,-48.131,-178.755,5.722,148.639
C06665=1210.329,87.768,-48.149,-178.753,5.723,148.639
C06666=1210.325,88.018,-48.167,-178.751,5.723,148.638
C06667=1210.320,88.267,-48.185,-178.747,5.725,148.638
C06668=1210.315,88.516,-48.203,-178.745,5.726,148.637
C06669=1210.310,88.765,-48.221,-178.743,5.726,148.637
C06670=1210.305,89.014,-48.239,-178.740,5.727,148.636
C06671=1210.300,89.264,-48.257,-178.737,5.729,148.636
C06672=1210.295,89.513,-48.275,-178.735,5.729,148.635
C06673=1210.291,89.763,-48.293,-178.733,5.730,148.634
C06674=1210.286,90.012,-48.311,-178.730,5.731,148.634
C06675=1210.281,90.261,-48.329,-178.727,5.732,148.633
C06676=1210.276,90.510,-48.347,-178.725,5.733,148.633
C06677=1210.271,90.759,-48.365,-178.722,5.734,148.632
C06678=1210.266,91.010,-48.384,-178.720,5.735,148.632
C06679=1210.261,91.259,-48.402,-178.717,5.736,148.631
C06680=1210.256,91.508,-48.420,-178.714,5.737,148.630
C06681=1210.252,91.757,-48.439,-178.712,5.737,148.630
C06682=1210.247,92.006,-48.457,-178.709,5.738,148.629
C06683=1210.243,92.256,-48.475,-178.706,5.739,148.629
C06684=1210.238,92.505,-48.493,-178.704,5.740,148.628
C06685=1210.233,92.754,-48.511,-178.701,5.741,148.628
C06686=1210.227,93.003,-48.530,-178.699,5.742,148.627
C06687=1210.222,93.253,-48.548,-178.696,5.743,148.627
C06688=1210.218,93.502,-48.567,-178.693,5.744,148.626
C06689=1210.213,93.751,-48.585,-178.691,5.745,148.625
C06690=1210.208,94.000,-48.603,-178.688,5.746,148.625
C06691=1210.203,94.250,-48.621,-178.686,5.747,148.624
C06692=1210.198,94.500,-48.640,-178.683,5.748,148.624
C06693=1210.194,94.748,-48.658,-178.681,5.748,148.623
C06694=1210.189,94.997,-48.676,-178.678,5.750,148.623
C06695=1210.184,95.246,-48.694,-178.675,5.751,148.622
C06696=1210.179,95.497,-48.713,-178.673,5.752,148.622
C06697=1210.174,95.745,-48.732,-178.670,5.753,148.621
C06698=1210.169,95.994,-48.750,-178.667,5.754,148.620
C06699=1210.165,96.244,-48.768,-178.665,5.755,148.620
C06700=1210.159,96.494,-48.787,-178.663,5.755,148.619
C06701=1210.155,96.742,-48.806,-178.660,5.757,148.619
C06702=1210.150,96.991,-48.824,-178.657,5.757,148.618
C06703=1210.146,97.241,-48.842,-178.655,5.758,148.618
C06704=1210.140,97.490,-48.861,-178.652,5.760,148.617
C06705=1210.135,97.739,-48.879,-178.649,5.760,148.617
C06706=1210.130,97.989,-48.897,-178.647,5.761,148.616
C06707=1210.126,98.238,-48.916,-178.645,5.762,148.615
C06708=1210.121,98.487,-48.935,-178.642,5.764,148.615
C06709=1210.116,98.737,-48.953,-178.639,5.764,148.614
C06710=1210.112,98.986,-48.972,-178.637,5.765,148.614
C06711=1210.106,99.235,-48.990,-178.634,5.767,148.613
C06712=1210.101,99.484,-49.008,-178.631,5.767,148.613
C06713=1210.097,99.734,-49.027,-178.629,5.768,148.612
C06714=1210.092,99.983,-49.046,-178.626,5.770,148.612
C06715=1210.087,100.232,-49.065,-178.624,5.770,148.611
C06716=1210.083,100.482,-49.083,-178.621,5.771,148.611
C06717=1210.077,100.731,-49.102,-178.618,5.772,148.610
C06718=1210.073,100.980,-49.120,-178.616,5.773,148.610
C06719=1210.068,101.230,-49.139,-178.613,5.774,148.609
C06720=1210.063,101.478,-49.158,-178.611,5.776,148.608
C06721=1210.058,101.728,-49.176,-178.608,5.776,148.608
C06722=1210.053,101.977,-49.196,-178.606,5.777,148.607
C06723=1210.048,102.226,-49.214,-178.603,5.778,148.607
C06724=1210.044,102.476,-49.233,-178.600,5.779,148.606
C06725=1210.039,102.725,-49.251,-178.598,5.780,148.606
C06726=1210.034,102.974,-49.270,-178.595,5.781,148.605
C06727=1210.029,103.224,-49.289,-178.593,5.783,148.605
C06728=1210.024,103.472,-49.308,-178.590,5.783,148.604
C06729=1210.019,103.722,-49.326,-178.588,5.784,148.604
C06730=1210.015,103.971,-49.345,-178.585,5.786,148.603
C06731=1210.010,104.220,-49.364,-178.583,5.787,148.603
C06732=1210.005,104.470,-49.383,-178.580,5.787,148.602
C06733=1210.000,104.718,-49.401,-178.577,5.789,148.601
C06734=1209.995,104.968,-49.420,-178.575,5.789,148.601
C06735=1209.991,105.217,-49.439,-178.572,5.791,148.600
C06736=1209.985,105.466,-49.458,-178.569,5.792,148.600
C06737=1209.981,105.716,-49.477,-178.567,5.792,148.599
C06738=1209.976,105.965,-49.496,-178.564,5.794,148.599
C06739=1209.972,106.215,-49.514,-178.562,5.795,148.598
C06740=1209.966,106.463,-49.534,-178.559,5.796,148.598
C06741=1209.962,106.713,-49.553,-178.556,5.797,148.597
C06742=1209.956,106.981,-49.573,-178.554,5.798,148.596
C06743=1209.951,107.249,-49.593,-178.551,5.799,148.596
C06744=1209.946,107.518,-49.613,-178.548,5.800,148.595
C06745=1209.941,107.786,-49.634,-178.545,5.802,148.595
C06746=1209.936,108.036,-49.654,-178.543,5.802,148.594
C06747=1209.931,108.284,-49.672,-178.540,5.803,148.594
C06748=1209.926,108.534,-49.691,-178.538,5.805,148.593
C06749=1209.922,108.783,-49.710,-178.535,5.805,148.593
C06750=1209.917,109.033,-49.730,-178.532,5.807,148.592
C06751=1209.911,109.282,-49.748,-178.530,5.808,148.592
C06752=1209.907,109.531,-49.767,-178.527,5.808,148.591
C06753=1209.902,109.780,-49.787,-178.524,5.810,148.591
C06754=1209.898,110.029,-49.806,-178.522,5.811,148.590
C06755=1209.893,110.278,-49.825,-178.520,5.812,148.589
C06756=1209.888,110.528,-49.843,-178.517,5.813,148.589
C06757=1209.883,110.777,-49.863,-178.514,5.814,148.588
C06758=1209.878,111.027,-49.882,-178.511,5.815,148.588
C06759=1209.874,111.275,-49.901,-178.509,5.816,148.587
C06760=1209.869,111.525,-49.921,-178.506,5.817,148.587
C06761=1209.864,111.774,-49.940,-178.504,5.819,148.586
C06762=1209.859,112.024,-49.958,-178.501,5.819,148.586
C06763=1209.854,112.272,-49.977,-178.499,5.820,148.585
C06764=1209.849,112.522,-49.997,-178.496,5.822,148.585
C06765=1209.845,112.771,-50.016,-178.494,5.823,148.584
C06766=1209.840,113.020,-50.035,-178.491,5.824,148.584
C06767=1209.835,113.269,-50.055,-178.488,5.825,148.583
C06768=1209.831,113.518,-50.074,-178.486,5.826,148.583
C06769=1209.826,113.768,-50.093,-178.483,5.827,148.582
C06770=1209.820,114.017,-50.113,-178.481,5.828,148.582
C06771=1209.816,114.266,-50.132,-178.478,5.830,148.581
C06772=1209.811,114.515,-50.151,-178.475,5.830,148.581
C06773=1209.806,114.764,-50.171,-178.473,5.831,148.580
C06774=1209.801,115.013,-50.190,-178.470,5.833,148.579
C06775=1209.797,115.262,-50.209,-178.468,5.834,148.579
C06776=1209.792,115.512,-50.229,-178.465,5.835,148.578
C06777=1209.787,115.761,-50.248,-178.462,5.836,148.578
C06778=1209.782,116.010,-50.268,-178.460,5.837,148.577
C06779=1209.778,116.259,-50.286,-178.457,5.838,148.577
C06780=1209.773,116.509,-50.306,-178.455,5.839,148.576
C06781=1209.768,116.758,-50.326,-178.452,5.841,148.576
C06782=1209.763,117.007,-50.345,-178.449,5.841,148.575
C06783=1209.758,117.257,-50.365,-178.447,5.842,148.575
C06784=1209.753,117.505,-50.383,-178.444,5.844,148.574
C06785=1209.749,117.755,-50.403,-178.442,5.845,148.574
C06786=1209.744,118.004,-50.423,-178.439,5.846,148.573
C06787=1209.739,118.253,-50.442,-178.437,5.847,148.573
C06788=1209.734,118.503,-50.462,-178.433,5.849,148.572
C06789=1209.730,118.752,-50.481,-178.431,5.850,148.572
C06790=1209.724,119.001,-50.500,-178.429,5.850,148.571
C06791=1209.720,119.250,-50.520,-178.426,5.852,148.571
C06792=1209.715,119.499,-50.540,-178.424,5.853,148.570
C06793=1209.710,119.748,-50.559,-178.421,5.854,148.570
C06794=1209.705,119.998,-50.579,-178.419,5.855,148.569
C06795=1209.701,120.247,-50.598,-178.415,5.857,148.569
C06796=1209.696,120.496,-50.617,-178.413,5.858,148.568
C06797=1209.691,120.745,-50.638,-178.411,5.858,148.568
C06798=1209.687,120.994,-50.657,-178.408,5.860,148.567
C06799=1209.681,121.243,-50.677,-178.405,5.861,148.567
C06800=1209.677,121.493,-50.696,-178.403,5.862,148.566
C06801=1209.672,121.742,-50.716,-178.400,5.863,148.566
C06802=1209.667,121.991,-50.736,-178.397,5.865,148.565
C06803=1209.662,122.240,-50.756,-178.395,5.866,148.565
C06804=1209.657,122.490,-50.775,-178.393,5.866,148.564
C06805=1209.653,122.739,-50.796,-178.390,5.868,148.564
C06806=1209.648,122.987,-50.814,-178.387,5.869,148.563
C06807=1209.644,123.237,-50.834,-178.385,5.870,148.563
C06808=1209.639,123.486,-50.854,-178.382,5.871,148.562
C06809=1209.634,123.735,-50.874,-178.379,5.873,148.562
C06810=1209.629,123.984,-50.893,-178.377,5.873,148.561
C06811=1209.624,124.234,-50.913,-178.374,5.875,148.561
C06812=1209.620,124.483,-50.933,-178.371,5.876,148.560
C06813=1209.614,124.732,-50.953,-178.369,5.878,148.560
C06814=1209.610,124.981,-50.972,-178.367,5.879,148.559
C06815=1209.605,125.230,-50.993,-178.364,5.879,148.559
C06816=1209.601,125.480,-51.012,-178.361,5.881,148.558
C06817=1209.596,125.728,-51.032,-178.359,5.882,148.558
C06818=1209.591,125.978,-51.052,-178.356,5.883,148.557
C06819=1209.586,126.227,-51.072,-178.353,5.884,148.557
C06820=1209.582,126.476,-51.092,-178.351,5.886,148.556
C06821=1209.577,126.726,-51.112,-178.349,5.887,148.556
C06822=1209.572,126.974,-51.132,-178.345,5.888,148.555
C06823=1209.567,127.223,-51.151,-178.343,5.889,148.555
C06824=1209.563,127.472,-51.172,-178.340,5.891,148.554
C06825=1209.558,127.722,-51.191,-178.338,5.892,148.554
C06826=1209.553,127.971,-51.212,-178.335,5.893,148.553
C06827=1209.547,128.220,-51.232,-178.333,5.894,148.553
C06828=1209.543,128.469,-51.252,-178.330,5.896,148.552
C06829=1209.538,128.719,-51.272,-178.327,5.896,148.552
C06830=1209.534,128.968,-51.292,-178.325,5.898,148.551
C06831=1209.529,129.217,-51.312,-178.322,5.899,148.551
C06832=1209.524,129.465,-51.332,-178.320,5.900,148.550
C06833=1209.519,129.715,-51.351,-178.317,5.901,148.550
C06834=1209.515,129.964,-51.372,-178.314,5.903,148.549
C06835=1209.510,130.213,-51.391,-178.312,5.904,148.549
C06836=1209.505,130.463,-51.412,-178.309,5.905,148.548
C06837=1209.500,130.712,-51.432,-178.307,5.906,148.548
C06838=1209.496,130.961,-51.452,-178.304,5.908,148.547
C06839=1209.491,131.209,-51.472,-178.302,5.909,148.547
C06840=1209.486,131.459,-51.492,-178.299,5.910,148.546
C06841=1209.481,131.708,-51.512,-178.296,5.911,148.546
C06842=1209.476,131.958,-51.533,-178.294,5.913,148.545
C06843=1209.472,132.207,-51.553,-178.291,5.913,148.545
C06844=1209.467,132.456,-51.573,-178.288,5.915,148.544
C06845=1209.462,132.705,-51.593,-178.286,5.916,148.544
C06846=1209.457,132.974,-51.615,-178.283,5.918,148.543
C06847=1209.452,133.242,-51.637,-178.280,5.918,148.543
C06848=1209.447,133.511,-51.659,-178.278,5.920,148.542
C06849=1209.441,133.780,-51.681,-178.275,5.921,148.542
C06850=1209.437,134.029,-51.701,-178.272,5.922,148.541
C06851=1209.432,134.278,-51.721,-178.270,5.924,148.541
C06852=1209.428,134.527,-51.741,-178.267,5.925,148.540
C06853=1209.422,134.776,-51.762,-178.264,5.927,148.540
C06854=1209.418,135.025,-51.782,-178.262,5.927,148.539
C06855=1209.413,135.274,-51.803,-178.259,5.929,148.539
C06856=1209.409,135.523,-51.823,-178.256,5.931,148.539
C06857=1209.403,135.772,-51.843,-178.254,5.931,148.538
C06858=1209.399,136.021,-51.863,-178.251,5.933,148.537
C06859=1209.394,136.270,-51.884,-178.249,5.934,148.537
C06860=1209.389,136.520,-51.905,-178.246,5.936,148.536
C06861=1209.384,136.769,-51.925,-178.244,5.937,148.536
C06862=1209.380,137.018,-51.945,-178.241,5.938,148.535
C06863=1209.375,137.267,-51.965,-178.239,5.939,148.535
C06864=1209.370,137.516,-51.986,-178.236,5.941,148.535
C06865=1209.366,137.765,-52.006,-178.233,5.941,148.534
C06866=1209.361,138.014,-52.027,-178.231,5.943,148.534
C06867=1209.356,138.263,-52.048,-178.228,5.944,148.533
C06868=1209.352,138.512,-52.068,-178.225,5.946,148.533
C06869=1209.346,138.762,-52.088,-178.223,5.947,148.532
C06870=1209.342,139.011,-52.109,-178.220,5.948,148.532
C06871=1209.337,139.260,-52.129,-178.217,5.950,148.531
C06872=1209.332,139.509,-52.150,-178.215,5.951,148.531
C06873=1209.328,139.758,-52.170,-178.212,5.952,148.530
C06874=1209.323,140.007,-52.191,-178.210,5.953,148.530
C06875=1209.318,140.257,-52.212,-178.207,5.955,148.529
C06876=1209.314,140.506,-52.232,-178.205,5.956,148.529
C06877=1209.308,140.755,-52.253,-178.202,5.957,148.528
C06878=1209.304,141.004,-52.274,-178.200,5.958,148.528
C06879=1209.299,141.253,-52.294,-178.197,5.960,148.527
C06880=1209.294,141.502,-52.315,-178.194,5.962,148.527
C06881=1209.290,141.751,-52.335,-178.192,5.962,148.527
C06882=1209.285,142.000,-52.356,-178.189,5.964,148.526
C06883=1209.280,142.249,-52.377,-178.187,5.965,148.526
C06884=1209.275,142.498,-52.398,-178.184,5.967,148.525
C06885=1209.271,142.747,-52.418,-178.181,5.967,148.525
C06886=1209.266,142.997,-52.439,-178.179,5.969,148.524
C06887=1209.262,143.246,-52.460,-178.176,5.971,148.524
C06888=1209.257,143.495,-52.481,-178.173,5.972,148.523
C06889=1209.252,143.744,-52.502,-178.171,5.973,148.523
C06890=1209.247,143.993,-52.523,-178.169,5.974,148.522
C06891=1209.243,144.242,-52.543,-178.165,5.976,148.522
C06892=1209.238,144.491,-52.564,-178.163,5.977,148.521
C06893=1209.233,144.740,-52.584,-178.161,5.978,148.521
C06894=1209.228,144.990,-52.605,-178.158,5.980,148.521
C06895=1209.224,145.238,-52.626,-178.155,5.981,148.520
C06896=1209.219,145.487,-52.647,-178.153,5.983,148.520
C06897=1209.214,145.736,-52.668,-178.150,5.983,148.519
C06898=1209.210,145.986,-52.689,-178.147,5.985,148.519
C06899=1209.205,146.235,-52.709,-178.145,5.987,148.518
C06900=1209.200,146.484,-52.730,-178.142,5.988,148.518
C06901=1209.195,146.733,-52.752,-178.139,5.989,148.517
C06902=1209.191,146.982,-52.772,-178.137,5.990,148.517
C06903=1209.186,147.231,-52.793,-178.134,5.992,148.516
C06904=1209.181,147.480,-52.814,-178.132,5.994,148.516
C06905=1209.176,147.729,-52.835,-178.129,5.994,148.516
C06906=1209.172,147.979,-52.857,-178.126,5.996,148.515
C06907=1209.167,148.228,-52.877,-178.124,5.997,148.515
C06908=1209.162,148.477,-52.898,-178.121,5.999,148.514
C06909=1209.158,148.725,-52.919,-178.119,6.001,148.514
C06910=1209.153,148.974,-52.940,-178.116,6.001,148.513
C06911=1209.148,149.224,-52.961,-178.114,6.003,148.513
C06912=1209.144,149.473,-52.983,-178.111,6.004,148.512
C06913=1209.139,149.722,-53.004,-178.108,6.005,148.512
C06914=1209.134,149.971,-53.025,-178.106,6.007,148.511
C06915=1209.130,150.220,-53.046,-178.104,6.008,148.511
C06916=1209.124,150.469,-53.067,-178.100,6.010,148.510
C06917=1209.120,150.717,-53.088,-178.098,6.011,148.510
C06918=1209.116,150.967,-53.109,-178.096,6.012,148.510
C06919=1209.111,151.216,-53.130,-178.093,6.014,148.509
C06920=1209.106,151.465,-53.152,-178.090,6.015,148.509
C06921=1209.101,151.714,-53.173,-178.088,6.017,148.508
C06922=1209.097,151.963,-53.194,-178.085,6.018,148.508
C06923=1209.092,152.213,-53.215,-178.082,6.019,148.507
C06924=1209.087,152.462,-53.236,-178.080,6.021,148.507
C06925=1209.082,152.710,-53.258,-178.077,6.023,148.507
C06926=1209.077,152.959,-53.278,-178.075,6.024,148.506
C06927=1209.073,153.209,-53.300,-178.072,6.025,148.506
C06928=1209.068,153.458,-53.321,-178.069,6.027,148.505
C06929=1209.063,153.707,-53.343,-178.067,6.028,148.505
C06930=1209.059,153.956,-53.363,-178.064,6.030,148.504
C06931=1209.054,154.205,-53.385,-178.062,6.030,148.504
C06932=1209.049,154.454,-53.406,-178.059,6.032,148.503
C06933=1209.044,154.703,-53.428,-178.056,6.034,148.503
C06934=1209.039,154.951,-53.450,-178.054,6.034,148.502
C06935=1209.036,155.201,-53.470,-178.051,6.036,148.502
C06936=1209.031,155.450,-53.492,-178.048,6.038,148.502
C06937=1209.026,155.699,-53.513,-178.046,6.039,148.501
C06938=1209.021,155.948,-53.535,-178.043,6.040,148.501
C06939=1209.016,156.198,-53.556,-178.040,6.042,148.500
C06940=1209.011,156.446,-53.578,-178.038,6.043,148.500
C06941=1209.007,156.695,-53.599,-178.036,6.045,148.500
C06942=1209.002,156.945,-53.620,-178.033,6.047,148.499
C06943=1208.998,157.193,-53.642,-178.030,6.047,148.499
C06944=1208.993,157.442,-53.663,-178.028,6.049,148.498
C06945=1208.988,157.692,-53.685,-178.025,6.051,148.498
C06946=1208.983,157.940,-53.706,-178.023,6.052,148.497
C06947=1208.978,158.189,-53.728,-178.020,6.054,148.497
C06948=1208.974,158.439,-53.749,-178.017,6.055,148.496
C06949=1208.969,158.688,-53.771,-178.015,6.056,148.496
C06950=1208.964,158.957,-53.794,-178.012,6.058,148.495
C06951=1208.959,159.225,-53.818,-178.009,6.060,148.495
C06952=1208.954,159.495,-53.841,-178.006,6.061,148.495
C06953=1208.949,159.764,-53.864,-178.003,6.063,148.494
C06954=1208.944,160.013,-53.886,-178.001,6.065,148.494
C06955=1208.940,160.262,-53.908,-177.999,6.066,148.493
C06956=1208.935,160.510,-53.929,-177.995,6.067,148.493
C06957=1208.930,160.760,-53.950,-177.993,6.069,148.492
C06958=1208.925,161.009,-53.972,-177.991,6.070,148.492
C06959=1208.921,161.258,-53.994,-177.988,6.072,148.492
C06960=1208.916,161.506,-54.016,-177.985,6.073,148.491
C06961=1208.911,161.756,-54.038,-177.983,6.074,148.491
C06962=1208.907,162.004,-54.060,-177.980,6.076,148.490
C06963=1208.902,162.254,-54.081,-177.977,6.078,148.490
C06964=1208.897,162.503,-54.103,-177.975,6.079,148.490
C06965=1208.892,162.752,-54.124,-177.972,6.080,148.489
C06966=1208.888,163.001,-54.146,-177.970,6.082,148.489
C06967=1208.883,163.250,-54.168,-177.967,6.084,148.488
C06968=1208.879,163.499,-54.190,-177.965,6.085,148.488
C06969=1208.874,163.748,-54.212,-177.962,6.087,148.487
C06970=1208.870,163.997,-54.234,-177.959,6.088,148.487
C06971=1208.865,164.246,-54.255,-177.957,6.089,148.486
C06972=1208.860,164.494,-54.277,-177.954,6.091,148.486
C06973=1208.855,164.744,-54.298,-177.952,6.093,148.486
C06974=1208.850,164.993,-54.320,-177.948,6.094,148.485
C06975=1208.846,165.242,-54.342,-177.946,6.095,148.485
C06976=1208.841,165.491,-54.364,-177.944,6.097,148.484
C06977=1208.837,165.740,-54.386,-177.941,6.099,148.484
C06978=1208.832,165.989,-54.408,-177.939,6.100,148.484
C06979=1208.827,166.238,-54.430,-177.936,6.101,148.483
C06980=1208.822,166.487,-54.452,-177.933,6.103,148.483
C06981=1208.818,166.736,-54.475,-177.930,6.105,148.482
C06982=1208.814,166.984,-54.496,-177.928,6.106,148.482
C06983=1208.809,167.234,-54.518,-177.926,6.107,148.482
C06984=1208.804,167.482,-54.540,-177.923,6.109,148.481
C06985=1208.800,167.731,-54.562,-177.920,6.110,148.481
C06986=1208.794,167.981,-54.584,-177.918,6.112,148.480
C06987=1208.790,168.229,-54.606,-177.915,6.114,148.480
C06988=1208.785,168.479,-54.628,-177.912,6.115,148.479
C06989=1208.780,168.727,-54.650,-177.910,6.116,148.479
C06990=1208.776,168.977,-54.672,-177.907,6.118,148.479
C06991=1208.771,169.226,-54.695,-177.904,6.120,148.478
C06992=1208.767,169.474,-54.717,-177.902,6.121,148.478
C06993=1208.762,169.724,-54.739,-177.900,6.122,148.477
C06994=1208.758,169.972,-54.761,-177.897,6.124,148.477
C06995=1208.753,170.222,-54.783,-177.894,6.126,148.477
C06996=1208.748,170.471,-54.805,-177.891,6.127,148.476
C06997=1208.744,170.719,-54.828,-177.889,6.128,148.476
C06998=1208.739,170.968,-54.849,-177.886,6.130,148.475
C06999=1208.735,171.217,-54.872,-177.884,6.132,148.475
C07000=1208.729,171.466,-54.894,-177.881,6.134,148.475
C07001=1208.725,171.716,-54.916,-177.879,6.135,148.474
C07002=1208.720,171.964,-54.938,-177.876,6.137,148.474
C07003=1208.715,172.213,-54.961,-177.873,6.138,148.473
C07004=1208.711,172.463,-54.983,-177.871,6.140,148.473
C07005=1208.706,172.711,-55.005,-177.868,6.141,148.473
C07006=1208.702,172.960,-55.027,-177.866,6.143,148.472
C07007=1208.696,173.209,-55.050,-177.863,6.145,148.472
C07008=1208.692,173.458,-55.072,-177.860,6.146,148.471
C07009=1208.688,173.707,-55.094,-177.857,6.148,148.471
C07010=1208.683,173.956,-55.117,-177.855,6.149,148.470
C07011=1208.679,174.205,-55.140,-177.853,6.151,148.470
C07012=1208.673,174.454,-55.162,-177.850,6.152,148.470
C07013=1208.669,174.703,-55.184,-177.847,6.154,148.469
C07014=1208.665,174.952,-55.207,-177.845,6.155,148.469
C07015=1208.659,175.201,-55.229,-177.842,6.157,148.469
C07016=1208.655,175.450,-55.251,-177.839,6.159,148.468
C07017=1208.650,175.698,-55.273,-177.837,6.160,148.468
C07018=1208.645,175.948,-55.296,-177.834,6.162,148.467
C07019=1208.641,176.196,-55.319,-177.832,6.163,148.467
C07020=1208.636,176.445,-55.341,-177.829,6.165,148.467
C07021=1208.632,176.694,-55.364,-177.827,6.167,148.466
C07022=1208.628,176.943,-55.386,-177.824,6.169,148.466
C07023=1208.622,177.192,-55.409,-177.822,6.170,148.466
C07024=1208.618,177.441,-55.431,-177.819,6.171,148.465
C07025=1208.613,177.690,-55.454,-177.816,6.173,148.465
C07026=1208.608,177.939,-55.476,-177.813,6.175,148.464
C07027=1208.604,178.188,-55.499,-177.811,6.176,148.464
C07028=1208.599,178.437,-55.521,-177.809,6.177,148.463
C07029=1208.594,178.685,-55.544,-177.806,6.179,148.463
C07030=1208.590,178.935,-55.566,-177.803,6.181,148.463
C07031=1208.585,179.184,-55.590,-177.801,6.183,148.462
C07032=1208.581,179.433,-55.612,-177.798,6.185,148.462
C07033=1208.576,179.681,-55.635,-177.795,6.186,148.461
C07034=1208.572,179.930,-55.658,-177.793,6.187,148.461
C07035=1208.567,180.180,-55.680,-177.790,6.189,148.461
C07036=1208.562,180.428,-55.703,-177.787,6.191,148.460
C07037=1208.557,180.677,-55.725,-177.785,6.193,148.460
C07038=1208.553,180.926,-55.748,-177.782,6.194,148.460
C07039=1208.548,181.175,-55.771,-177.780,6.195,148.459
C07040=1208.544,181.424,-55.793,-177.777,6.197,148.459
C07041=1208.539,181.673,-55.816,-177.775,6.199,148.459
C07042=1208.535,181.922,-55.839,-177.772,6.201,148.458
C07043=1208.530,182.171,-55.862,-177.769,6.202,148.458
C07044=1208.525,182.419,-55.884,-177.766,6.204,148.457
C07045=1208.521,182.668,-55.908,-177.764,6.205,148.457
C07046=1208.516,182.918,-55.930,-177.761,6.207,148.457
C07047=1208.512,183.167,-55.953,-177.759,6.209,148.456
C07048=1208.506,183.415,-55.976,-177.756,6.211,148.456
C07049=1208.502,183.664,-55.999,-177.753,6.212,148.455
C07050=1208.497,183.913,-56.021,-177.751,6.214,148.455
C07051=1208.493,184.162,-56.045,-177.749,6.215,148.455
C07052=1208.489,184.411,-56.067,-177.746,6.217,148.454
C07053=1208.483,184.659,-56.090,-177.743,6.219,148.454
C07054=1208.478,184.929,-56.115,-177.740,6.220,148.453
C07055=1208.473,185.199,-56.140,-177.738,6.222,148.453
C07056=1208.468,185.468,-56.165,-177.735,6.224,148.453
C07057=1208.464,185.738,-56.189,-177.732,6.226,148.452
C07058=1208.459,185.987,-56.213,-177.730,6.228,148.452
C07059=1208.454,186.236,-56.236,-177.727,6.229,148.452
C07060=1208.449,186.485,-56.259,-177.724,6.231,148.451
C07061=1208.446,186.734,-56.282,-177.721,6.233,148.451
C07062=1208.441,186.983,-56.306,-177.719,6.235,148.450
C07063=1208.435,187.232,-56.328,-177.716,6.236,148.450
C07064=1208.431,187.480,-56.351,-177.714,6.237,148.450
C07065=1208.427,187.729,-56.374,-177.711,6.239,148.449
C07066=1208.422,187.979,-56.397,-177.708,6.241,148.449
C07067=1208.417,188.228,-56.421,-177.706,6.243,148.449
C07068=1208.413,188.476,-56.443,-177.703,6.245,148.448
C07069=1208.408,188.725,-56.467,-177.701,6.247,148.448
C07070=1208.403,188.974,-56.490,-177.698,6.248,148.448
C07071=1208.398,189.223,-56.513,-177.695,6.250,148.447
C07072=1208.395,189.471,-56.536,-177.693,6.251,148.447
C07073=1208.390,189.720,-56.559,-177.690,6.253,148.446
C07074=1208.385,189.969,-56.583,-177.688,6.255,148.446
C07075=1208.380,190.218,-56.606,-177.685,6.257,148.446
C07076=1208.376,190.468,-56.629,-177.683,6.258,148.445
C07077=1208.371,190.717,-56.653,-177.680,6.260,148.445
C07078=1208.367,190.965,-56.676,-177.677,6.262,148.445
C07079=1208.362,191.214,-56.699,-177.675,6.264,148.444
C07080=1208.357,191.463,-56.722,-177.672,6.265,148.444
C07081=1208.353,191.711,-56.746,-177.670,6.267,148.444
C07082=1208.348,191.960,-56.769,-177.667,6.269,148.443
C07083=1208.343,192.209,-56.793,-177.664,6.270,148.443
C07084=1208.339,192.458,-56.815,-177.662,6.272,148.443
C07085=1208.335,192.707,-56.839,-177.659,6.274,148.442
C07086=1208.330,192.956,-56.862,-177.656,6.275,148.442
C07087=1208.325,193.205,-56.886,-177.653,6.277,148.441
C07088=1208.321,193.453,-56.910,-177.651,6.279,148.441
C07089=1208.316,193.702,-56.933,-177.648,6.281,148.441
C07090=1208.311,193.951,-56.956,-177.646,6.282,148.440
C07091=1208.307,194.200,-56.980,-177.643,6.284,148.440
C07092=1208.302,194.449,-57.003,-177.641,6.286,148.440
C07093=1208.298,194.698,-57.027,-177.638,6.287,148.439
C07094=1208.293,194.947,-57.050,-177.635,6.289,148.439
C07095=1208.288,195.196,-57.074,-177.633,6.291,148.439
C07096=1208.284,195.445,-57.097,-177.630,6.293,148.438
C07097=1208.280,195.693,-57.121,-177.627,6.295,148.438
C07098=1208.275,195.942,-57.144,-177.625,6.297,148.438
C07099=1208.270,196.191,-57.167,-177.622,6.298,148.437
C07100=1208.266,196.440,-57.191,-177.620,6.300,148.437
C07101=1208.261,196.689,-57.215,-177.617,6.301,148.436
C07102=1208.257,196.938,-57.238,-177.615,6.303,148.436
C07103=1208.252,197.187,-57.262,-177.612,6.305,148.436
C07104=1208.248,197.435,-57.286,-177.609,6.307,148.435
C07105=1208.243,197.684,-57.309,-177.607,6.308,148.435
C07106=1208.238,197.933,-57.334,-177.604,6.310,148.435
C07107=1208.233,198.182,-57.357,-177.602,6.312,148.434
C07108=1208.228,198.431,-57.380,-177.599,6.314,148.434
C07109=1208.224,198.679,-57.404,-177.596,6.316,148.434
C07110=1208.219,198.928,-57.428,-177.594,6.318,148.434
C07111=1208.215,199.177,-57.452,-177.591,6.320,148.433
C07112=1208.210,199.426,-57.475,-177.589,6.322,148.433
C07113=1208.205,199.675,-57.499,-177.586,6.323,148.433
C07114=1208.201,199.923,-57.523,-177.583,6.325,148.432
C07115=1208.196,200.172,-57.546,-177.581,6.327,148.432
C07116=1208.192,200.421,-57.570,-177.578,6.329,148.432
C07117=1208.187,200.670,-57.593,-177.576,6.331,148.431
C07118=1208.183,200.919,-57.618,-177.573,6.332,148.431
C07119=1208.178,201.168,-57.642,-177.571,6.334,148.430
C07120=1208.174,201.417,-57.666,-177.568,6.335,148.430
C07121=1208.169,201.666,-57.689,-177.565,6.337,148.430
C07122=1208.165,201.914,-57.713,-177.563,6.339,148.429
C07123=1208.160,202.163,-57.737,-177.560,6.341,148.429
C07124=1208.155,202.411,-57.761,-177.558,6.343,148.429
C07125=1208.151,202.660,-57.785,-177.555,6.345,148.428
C07126=1208.146,202.909,-57.809,-177.552,6.346,148.428
C07127=1208.142,203.158,-57.833,-177.550,6.348,148.428
C07128=1208.137,203.407,-57.857,-177.547,6.350,148.427
C07129=1208.133,203.656,-57.881,-177.544,6.352,148.427
C07130=1208.128,203.904,-57.905,-177.542,6.354,148.427
C07131=1208.123,204.154,-57.929,-177.539,6.356,148.426
C07132=1208.119,204.402,-57.953,-177.536,6.357,148.426
C07133=1208.114,204.650,-57.977,-177.534,6.359,148.426
C07134=1208.110,204.900,-58.001,-177.531,6.361,148.425
C07135=1208.106,205.149,-58.025,-177.529,6.363,148.425
C07136=1208.100,205.397,-58.049,-177.526,6.365,148.425
C07137=1208.096,205.646,-58.073,-177.524,6.367,148.425
C07138=1208.091,205.895,-58.097,-177.521,6.369,148.424
C07139=1208.086,206.143,-58.121,-177.518,6.370,148.424
C07140=1208.082,206.393,-58.146,-177.516,6.372,148.424
C07141=1208.078,206.642,-58.169,-177.513,6.374,148.423
C07142=1208.073,206.890,-58.193,-177.510,6.376,148.423
C07143=1208.068,207.139,-58.218,-177.508,6.378,148.422
C07144=1208.064,207.387,-58.242,-177.505,6.380,148.422
C07145=1208.060,207.637,-58.266,-177.502,6.381,148.422
C07146=1208.055,207.886,-58.290,-177.500,6.383,148.421
C07147=1208.050,208.134,-58.314,-177.497,6.385,148.421
C07148=1208.046,208.382,-58.339,-177.495,6.387,148.421
C07149=1208.041,208.632,-58.364,-177.492,6.389,148.421
C07150=1208.037,208.880,-58.388,-177.490,6.391,148.420
C07151=1208.032,209.129,-58.411,-177.487,6.393,148.420
C07152=1208.027,209.378,-58.436,-177.484,6.395,148.420
C07153=1208.023,209.627,-58.460,-177.482,6.396,148.419
C07154=1208.018,209.876,-58.485,-177.479,6.398,148.419
C07155=1208.014,210.124,-58.509,-177.476,6.400,148.419
C07156=1208.009,210.373,-58.533,-177.474,6.402,148.418
C07157=1208.005,210.622,-58.558,-177.471,6.404,148.418
C07158=1208.000,210.892,-58.585,-177.469,6.406,148.418
C07159=1207.995,211.163,-58.610,-177.466,6.407,148.417
C07160=1207.990,211.433,-58.637,-177.463,6.410,148.417
C07161=1207.985,211.703,-58.664,-177.460,6.412,148.417
C07162=1207.981,211.952,-58.688,-177.457,6.414,148.416
C07163=1207.976,212.201,-58.713,-177.455,6.416,148.416
C07164=1207.971,212.449,-58.737,-177.452,6.417,148.416
C07165=1207.967,212.699,-58.762,-177.450,6.420,148.416
C07166=1207.962,212.947,-58.786,-177.447,6.421,148.415
C07167=1207.957,213.196,-58.811,-177.445,6.423,148.415
C07168=1207.953,213.445,-58.835,-177.442,6.425,148.415
C07169=1207.948,213.694,-58.860,-177.439,6.427,148.414
C07170=1207.944,213.942,-58.884,-177.437,6.429,148.414
C07171=1207.939,214.192,-58.909,-177.434,6.431,148.414
C07172=1207.935,214.440,-58.933,-177.432,6.432,148.413
C07173=1207.930,214.688,-58.958,-177.429,6.434,148.413
C07174=1207.926,214.937,-58.983,-177.426,6.437,148.413
C07175=1207.921,215.186,-59.007,-177.423,6.439,148.412
C07176=1207.917,215.434,-59.031,-177.421,6.441,148.412
C07177=1207.912,215.684,-59.056,-177.418,6.443,148.412
C07178=1207.907,215.932,-59.081,-177.416,6.445,148.411
C07179=1207.903,216.181,-59.105,-177.413,6.446,148.411
C07180=1207.899,216.430,-59.131,-177.410,6.448,148.411
C07181=1207.894,216.678,-59.155,-177.408,6.450,148.411
C07182=1207.890,216.928,-59.180,-177.405,6.452,148.410
C07183=1207.885,217.176,-59.204,-177.403,6.454,148.410
C07184=1207.880,217.424,-59.229,-177.400,6.456,148.410
C07185=1207.876,217.673,-59.255,-177.398,6.458,148.409
C07186=1207.872,217.922,-59.279,-177.395,6.460,148.409
C07187=1207.867,218.171,-59.304,-177.392,6.462,148.409
C07188=1207.862,218.419,-59.329,-177.390,6.464,148.409
C07189=1207.858,218.668,-59.353,-177.388,6.466,148.408
C07190=1207.853,218.917,-59.378,-177.385,6.467,148.408
C07191=1207.848,219.165,-59.403,-177.382,6.470,148.408
C07192=1207.845,219.414,-59.428,-177.379,6.472,148.407
C07193=1207.840,219.663,-59.453,-177.376,6.474,148.407
C07194=1207.835,219.912,-59.478,-177.374,6.476,148.407
C07195=1207.831,220.160,-59.502,-177.372,6.478,148.407
C07196=1207.826,220.409,-59.527,-177.369,6.480,148.406
C07197=1207.822,220.658,-59.553,-177.366,6.481,148.406
C07198=1207.817,220.906,-59.577,-177.364,6.483,148.406
C07199=1207.813,221.156,-59.602,-177.361,6.485,148.405
C07200=1207.808,221.404,-59.627,-177.359,6.487,148.405
C07201=1207.804,221.653,-59.652,-177.356,6.489,148.405
C07202=1207.799,221.901,-59.677,-177.354,6.491,148.404
C07203=1207.795,222.150,-59.702,-177.351,6.493,148.404
C07204=1207.790,222.399,-59.728,-177.348,6.495,148.404
C07205=1207.786,222.648,-59.752,-177.346,6.498,148.404
C07206=1207.781,222.896,-59.777,-177.343,6.499,148.403
C07207=1207.777,223.145,-59.802,-177.340,6.501,148.403
C07208=1207.772,223.393,-59.828,-177.338,6.503,148.403
C07209=1207.767,223.643,-59.853,-177.335,6.505,148.402
C07210=1207.763,223.891,-59.878,-177.333,6.507,148.402
C07211=1207.759,224.140,-59.903,-177.330,6.509,148.402
C07212=1207.754,224.388,-59.928,-177.328,6.511,148.402
C07213=1207.749,224.638,-59.953,-177.325,6.513,148.401
C07214=1207.745,224.886,-59.978,-177.322,6.514,148.401
C07215=1207.740,225.135,-60.004,-177.320,6.517,148.401
C07216=1207.736,225.383,-60.028,-177.317,6.519,148.401
C07217=1207.732,225.632,-60.054,-177.314,6.521,148.400
C07218=1207.727,225.880,-60.079,-177.312,6.523,148.400
C07219=1207.722,226.129,-60.104,-177.309,6.525,148.400
C07220=1207.718,226.379,-60.130,-177.307,6.527,148.399
C07221=1207.713,226.627,-60.155,-177.304,6.529,148.399
C07222=1207.709,226.875,-60.181,-177.302,6.531,148.399
C07223=1207.704,227.124,-60.205,-177.299,6.533,148.399
C07224=1207.700,227.373,-60.230,-177.297,6.535,148.398
C07225=1207.695,227.621,-60.256,-177.294,6.537,148.398
C07226=1207.691,227.870,-60.282,-177.291,6.539,148.398
C07227=1207.687,228.119,-60.307,-177.288,6.541,148.397
C07228=1207.682,228.367,-60.332,-177.286,6.543,148.397
C07229=1207.677,228.616,-60.358,-177.284,6.545,148.397
C07230=1207.672,228.865,-60.382,-177.281,6.547,148.397
C07231=1207.668,229.113,-60.408,-177.278,6.549,148.396
C07232=1207.664,229.362,-60.434,-177.276,6.551,148.396
C07233=1207.659,229.610,-60.459,-177.274,6.553,148.396
C07234=1207.655,229.859,-60.485,-177.271,6.555,148.396
C07235=1207.650,230.109,-60.510,-177.268,6.557,148.395
C07236=1207.645,230.357,-60.536,-177.266,6.560,148.395
C07237=1207.641,230.606,-60.561,-177.263,6.561,148.395
C07238=1207.636,230.854,-60.587,-177.260,6.563,148.395
C07239=1207.632,231.102,-60.612,-177.258,6.565,148.394
C07240=1207.628,231.351,-60.638,-177.256,6.567,148.394
C07241=1207.623,231.600,-60.663,-177.253,6.569,148.394
C07242=1207.619,231.849,-60.689,-177.250,6.571,148.394
C07243=1207.614,232.098,-60.714,-177.247,6.574,148.393
C07244=1207.610,232.346,-60.740,-177.245,6.576,148.393
C07245=1207.605,232.594,-60.765,-177.242,6.578,148.393
C07246=1207.601,232.843,-60.791,-177.240,6.579,148.393
C07247=1207.596,233.091,-60.817,-177.238,6.582,148.392
C07248=1207.592,233.340,-60.842,-177.235,6.583,148.392
C07249=1207.587,233.589,-60.869,-177.232,6.585,148.392
C07250=1207.582,233.837,-60.894,-177.229,6.588,148.391
C07251=1207.578,234.086,-60.920,-177.227,6.590,148.391
C07252=1207.574,234.335,-60.946,-177.224,6.592,148.391
C07253=1207.570,234.584,-60.971,-177.222,6.594,148.391
C07254=1207.565,234.832,-60.997,-177.220,6.596,148.391
C07255=1207.561,235.081,-61.022,-177.217,6.598,148.390
C07256=1207.556,235.330,-61.048,-177.214,6.600,148.390
C07257=1207.551,235.578,-61.074,-177.211,6.602,148.390
C07258=1207.547,235.827,-61.100,-177.209,6.605,148.390
C07259=1207.542,236.076,-61.126,-177.206,6.606,148.389
C07260=1207.538,236.324,-61.151,-177.204,6.608,148.389
C07261=1207.533,236.572,-61.177,-177.201,6.610,148.389
C07262=1207.529,236.844,-61.206,-177.198,6.613,148.389
C07263=1207.524,237.116,-61.234,-177.196,6.615,148.388
C07264=1207.518,237.387,-61.263,-177.192,6.618,148.388
C07265=1207.514,237.658,-61.291,-177.190,6.620,148.388
C07266=1207.510,237.907,-61.316,-177.188,6.622,148.388
C07267=1207.505,238.156,-61.342,-177.185,6.624,148.387
C07268=1207.501,238.404,-61.368,-177.182,6.626,148.387
C07269=1207.496,238.653,-61.395,-177.180,6.628,148.387
C07270=1207.492,238.901,-61.420,-177.177,6.630,148.387
C07271=1207.487,239.150,-61.446,-177.174,6.632,148.386
C07272=1207.483,239.399,-61.472,-177.172,6.634,148.386
C07273=1207.478,239.647,-61.499,-177.170,6.636,148.386
C07274=1207.474,239.896,-61.524,-177.167,6.639,148.386
C07275=1207.469,240.144,-61.550,-177.164,6.641,148.385
C07276=1207.464,240.394,-61.576,-177.162,6.643,148.385
C07277=1207.461,240.642,-61.603,-177.159,6.645,148.385
C07278=1207.456,240.890,-61.628,-177.157,6.647,148.385
C07279=1207.451,241.139,-61.655,-177.154,6.649,148.384
C07280=1207.447,241.387,-61.681,-177.151,6.651,148.384
C07281=1207.443,241.636,-61.707,-177.149,6.654,148.384
C07282=1207.438,241.885,-61.733,-177.146,6.655,148.384
C07283=1207.434,242.133,-61.760,-177.144,6.658,148.384
C07284=1207.429,242.381,-61.785,-177.142,6.659,148.383
C07285=1207.424,242.630,-61.811,-177.138,6.662,148.383
C07286=1207.420,242.879,-61.838,-177.136,6.664,148.383
C07287=1207.416,243.127,-61.864,-177.134,6.666,148.383
C07288=1207.411,243.376,-61.891,-177.131,6.668,148.382
C07289=1207.407,243.625,-61.916,-177.129,6.670,148.382
C07290=1207.402,243.874,-61.943,-177.126,6.673,148.382
C07291=1207.398,244.122,-61.969,-177.123,6.675,148.382
C07292=1207.393,244.370,-61.995,-177.121,6.677,148.382
C07293=1207.389,244.619,-62.022,-177.118,6.679,148.381
C07294=1207.384,244.867,-62.047,-177.116,6.681,148.381
C07295=1207.380,245.116,-62.074,-177.113,6.684,148.381
C07296=1207.375,245.365,-62.100,-177.110,6.685,148.381
C07297=1207.371,245.613,-62.127,-177.108,6.688,148.380
C07298=1207.367,245.862,-62.153,-177.106,6.689,148.380
C07299=1207.362,246.111,-62.180,-177.103,6.692,148.380
C07300=1207.358,246.359,-62.206,-177.100,6.694,148.380
C07301=1207.353,246.608,-62.233,-177.098,6.696,148.379
C07302=1207.349,246.856,-62.259,-177.095,6.698,148.379
C07303=1207.344,247.105,-62.286,-177.093,6.700,148.379
C07304=1207.340,247.353,-62.312,-177.090,6.703,148.379
C07305=1207.335,247.602,-62.339,-177.087,6.705,148.379
C07306=1207.331,247.850,-62.365,-177.085,6.707,148.378
C07307=1207.326,248.098,-62.392,-177.083,6.709,148.378
C07308=1207.322,248.347,-62.417,-177.080,6.712,148.378
C07309=1207.317,248.596,-62.444,-177.077,6.714,148.378
C07310=1207.313,248.844,-62.471,-177.075,6.716,148.378
C07311=1207.308,249.093,-62.497,-177.072,6.718,148.377
C07312=1207.304,249.342,-62.524,-177.070,6.720,148.377
C07313=1207.300,249.590,-62.551,-177.067,6.723,148.377
C07314=1207.295,249.839,-62.577,-177.065,6.725,148.377
C07315=1207.291,250.087,-62.604,-177.062,6.727,148.376
